SPLINE
SPL {X  -162.820, Y  +621.304, Z    +0.000, E1   +22.259, E3 +517644.135}
SPL {X  -162.820, Y  +618.758, Z    +0.000, E1   +22.239, E3 +517657.285}
SPL {X  -162.820, Y  +616.062, Z    +0.000, E1   +22.275, E3 +517670.706}
SPL {X  -162.820, Y  +613.536, Z    +0.000, E1   +22.242, E3 +517683.827}
SPL {X  -162.820, Y  +611.128, Z    +0.000, E1   +22.252, E3 +517695.998}
SPL {X  -162.820, Y  +608.428, Z    +0.000, E1   +22.255, E3 +517709.782}
SPL {X  -162.820, Y  +605.178, Z    +0.000, E1   +22.267, E3 +517726.314}
SPL {X  -162.820, Y  +602.350, Z    +0.000, E1   +22.224, E3 +517740.931}
SPL {X  -162.820, Y  +599.168, Z    +0.000, E1   +22.310, E3 +517756.585}
SPL {X  -162.820, Y  +595.597, Z    +0.000, E1   +22.284, E3 +517774.921}
SPL {X  -162.820, Y  +593.320, Z    +0.000, E1   +22.199, E3 +517787.011}
SPL {X  -162.820, Y  +591.031, Z    +0.000, E1   +22.283, E3 +517798.102}
SPL {X  -162.820, Y  +588.026, Z    +0.000, E1   +22.301, E3 +517813.229}
SPL {X  -162.820, Y  +585.899, Z    +0.000, E1   +22.286, E3 +517824.031}
SPL {X  -162.820, Y  +583.204, Z    +0.000, E1   +22.278, E3 +517838.054}
SPL {X  -162.820, Y  +580.317, Z    +0.000, E1   +22.300, E3 +517852.325}
SPL {X  -162.820, Y  +578.061, Z    +0.000, E1   +22.264, E3 +517864.210}
SPL {X  -162.820, Y  +575.394, Z    +0.000, E1   +22.240, E3 +517877.954}
SPL {X  -162.820, Y  +573.156, Z    +0.000, E1   +22.254, E3 +517889.164}
SPL {X  -162.820, Y  +570.852, Z    +0.000, E1   +22.234, E3 +517901.188}
SPL {X  -162.820, Y  +568.608, Z    +0.000, E1   +22.253, E3 +517912.321}
SPL {X  -162.820, Y  +565.838, Z    +0.000, E1   +22.271, E3 +517926.553}
SPL {X  -162.820, Y  +562.162, Z    +0.000, E1   +22.252, E3 +517945.370}
SPL {X  -162.820, Y  +559.515, Z    +0.000, E1   +22.273, E3 +517958.488}
SPL {X  -162.820, Y  +556.723, Z    +0.000, E1   +22.309, E3 +517972.572}
SPL {X  -162.820, Y  +553.294, Z    +0.000, E1   +22.266, E3 +517990.360}
SPL {X  -162.820, Y  +550.136, Z    +0.000, E1   +22.258, E3 +518006.473}
SPL {X  -162.820, Y  +546.694, Z    +0.000, E1   +22.290, E3 +518023.795}
SPL {X  -162.820, Y  +543.558, Z    +0.000, E1   +22.285, E3 +518039.658}
SPL {X  -162.820, Y  +541.633, Z    +0.000, E1   +22.257, E3 +518049.586}
SPL {X  -162.820, Y  +539.116, Z    +0.000, E1   +22.302, E3 +518062.197}
SPL {X  -162.820, Y  +536.913, Z    +0.000, E1   +22.192, E3 +518074.121}
SPL {X  -162.820, Y  +534.880, Z    +0.000, E1   +22.252, E3 +518084.075}
SPL {X  -162.820, Y  +532.896, Z    +0.000, E1   +22.234, E3 +518094.235}
SPL {X  -162.820, Y  +531.056, Z    +0.000, E1   +22.251, E3 +518103.517}
SPL {X  -162.820, Y  +528.708, Z    +0.000, E1   +22.319, E3 +518114.899}
SPL {X  -162.820, Y  +525.932, Z    +0.000, E1   +22.258, E3 +518129.655}
SPL {X  -162.820, Y  +522.524, Z    +0.000, E1   +22.326, E3 +518146.379}
SPL {X  -162.820, Y  +519.457, Z    +0.000, E1   +22.481, E3 +518160.508}
SPL {X  -162.820, Y  +505.859, Z    +0.000, E1   +28.367, E3 +518174.991}
SPL {X  -162.820, Y  +504.131, Z    +0.000, E1   +27.325, E3 +518189.129}
SPL {X  -162.820, Y  +503.215, Z    +0.000, E1   +26.369, E3 +518199.815}
SPL {X  -162.820, Y  +502.502, Z    +0.000, E1   +25.597, E3 +518208.662}
SPL {X  -162.820, Y  +501.672, Z    +0.000, E1   +24.583, E3 +518220.277}
SPL {X  -162.820, Y  +500.515, Z    +0.000, E1   +23.444, E3 +518234.807}
SPL {X  -162.820, Y  +499.633, Z    +0.000, E1   +22.486, E3 +518246.853}
SPL {X  -162.820, Y  +498.303, Z    +0.000, E1   +21.749, E3 +518260.163}
SPL {X  -162.820, Y  +495.897, Z    +0.000, E1   +21.662, E3 +518273.316}
SPL {X  -162.820, Y  +493.717, Z    +0.000, E1   +21.704, E3 +518284.422}
SPL {X  -162.820, Y  +491.396, Z    +0.000, E1   +21.707, E3 +518296.546}
SPL {X  -162.820, Y  +489.485, Z    +0.000, E1   +21.661, E3 +518306.894}
SPL {X  -162.820, Y  +487.723, Z    +0.000, E1   +21.665, E3 +518316.098}
SPL {X  -162.820, Y  +485.661, Z    +0.000, E1   +21.712, E3 +518326.541}
SPL {X  -162.820, Y  +482.775, Z    +0.000, E1   +21.716, E3 +518341.794}
SPL {X  -162.820, Y  +479.894, Z    +0.000, E1   +21.695, E3 +518356.870}
SPL {X  -162.820, Y  +477.685, Z    +0.000, E1   +21.656, E3 +518368.807}
SPL {X  -162.820, Y  +475.419, Z    +0.000, E1   +21.711, E3 +518380.160}
SPL {X  -162.820, Y  +473.301, Z    +0.000, E1   +21.712, E3 +518391.257}
SPL {X  -162.820, Y  +470.965, Z    +0.000, E1   +21.700, E3 +518403.602}
SPL {X  -162.820, Y  +469.036, Z    +0.000, E1   +21.695, E3 +518413.646}
SPL {X  -162.820, Y  +467.138, Z    +0.000, E1   +21.678, E3 +518423.817}
SPL {X  -162.820, Y  +465.011, Z    +0.000, E1   +21.692, E3 +518434.800}
SPL {X  -162.820, Y  +462.669, Z    +0.000, E1   +21.752, E3 +518446.580}
SPL {X  -162.820, Y  +460.725, Z    +0.000, E1   +21.689, E3 +518457.193}
SPL {X  -162.820, Y  +458.666, Z    +0.000, E1   +21.695, E3 +518468.005}
SPL {X  -162.820, Y  +456.431, Z    +0.000, E1   +21.708, E3 +518479.534}
SPL {X  -162.820, Y  +454.628, Z    +0.000, E1   +21.674, E3 +518489.252}
SPL {X  -162.820, Y  +452.690, Z    +0.000, E1   +21.773, E3 +518498.526}
SPL {X  -162.820, Y  +450.610, Z    +0.000, E1   +21.698, E3 +518510.125}
SPL {X  -162.820, Y  +448.170, Z    +0.000, E1   +21.667, E3 +518523.146}
SPL {X  -162.820, Y  +446.246, Z    +0.000, E1   +21.696, E3 +518532.964}
SPL {X  -162.820, Y  +443.784, Z    +0.000, E1   +21.713, E3 +518545.750}
SPL {X  -162.820, Y  +441.754, Z    +0.000, E1   +21.708, E3 +518556.302}
SPL {X  -162.820, Y  +439.933, Z    +0.000, E1   +21.690, E3 +518566.066}
SPL {X  -162.820, Y  +437.628, Z    +0.000, E1   +21.678, E3 +518578.254}
SPL {X  -162.820, Y  +434.473, Z    +0.000, E1   +21.747, E3 +518594.350}
SPL {X  -162.820, Y  +431.492, Z    +0.000, E1   +21.686, E3 +518610.299}
SPL {X  -162.820, Y  +429.074, Z    +0.000, E1   +21.710, E3 +518622.751}
SPL {X  -162.820, Y  +426.023, Z    +0.000, E1   +21.718, E3 +518638.819}
SPL {X  -162.820, Y  +422.986, Z    +0.000, E1   +21.685, E3 +518654.866}
SPL {X  -162.820, Y  +420.528, Z    +0.000, E1   +21.706, E3 +518667.516}
SPL {X  -162.820, Y  +418.116, Z    +0.000, E1   +21.761, E3 +518679.663}
SPL {X  -162.820, Y  +416.127, Z    +0.000, E1   +21.715, E3 +518690.368}
SPL {X  -162.820, Y  +414.361, Z    +0.000, E1   +21.613, E3 +518700.556}
SPL {X  -162.820, Y  +411.450, Z    +0.000, E1   +21.710, E3 +518715.129}
SPL {X  -162.820, Y  +408.590, Z    +0.000, E1   +21.735, E3 +518729.755}
SPL {X  -162.820, Y  +406.238, Z    +0.000, E1   +21.697, E3 +518742.404}
SPL {X  -162.820, Y  +403.166, Z    +0.000, E1   +21.746, E3 +518758.209}
SPL {X  -162.820, Y  +400.348, Z    +0.000, E1   +21.713, E3 +518773.044}
SPL {X  -162.820, Y  +398.298, Z    +0.000, E1   +21.721, E3 +518783.660}
SPL {X  -162.820, Y  +396.371, Z    +0.000, E1   +21.713, E3 +518793.842}
SPL {X  -162.820, Y  +394.508, Z    +0.000, E1   +21.616, E3 +518804.397}
SPL {X  -162.820, Y  +391.777, Z    +0.000, E1   +21.714, E3 +518818.057}
SPL {X  -162.820, Y  +388.822, Z    +0.000, E1   +21.717, E3 +518833.376}
SPL {X  -162.820, Y  +386.818, Z    +0.000, E1   +21.679, E3 +518844.116}
SPL {X  -162.820, Y  +384.697, Z    +0.000, E1   +21.693, E3 +518855.186}
SPL {X  -162.820, Y  +382.288, Z    +0.000, E1   +21.742, E3 +518867.310}
SPL {X  -162.817, Y  +379.520, Z    +0.000, E1   +21.723, E3 +518882.147}
SPL {X  -162.776, Y  +376.710, Z    +0.000, E1   +21.698, E3 +518896.887}
SPL {X  -162.707, Y  +374.438, Z    +0.000, E1   +21.688, E3 +518908.890}
SPL {X  -162.607, Y  +372.171, Z    +0.000, E1   +21.692, E3 +518920.690}
SPL {X  -162.494, Y  +370.197, Z    +0.000, E1   +21.655, E3 +518931.316}
SPL {X  -162.349, Y  +368.131, Z    +0.000, E1   +21.624, E3 +518942.434}
SPL {X  -162.161, Y  +365.866, Z    +0.000, E1   +21.642, E3 +518954.120}
SPL {X  -161.927, Y  +363.466, Z    +0.000, E1   +21.730, E3 +518965.891}
SPL {X  -160.290, Y  +351.907, Z    +0.000, E1   +27.562, E3 +518973.469}
SPL {X  -159.725, Y  +348.905, Z    +0.000, E1   +26.136, E3 +518998.704}
ENDSPLINE

SPLINE
SPL {X  -160.871, Y  +355.385, Z    +0.000, E1   +21.841, E3 +519007.547}
SPL {X  -161.833, Y  +362.603, Z    +0.000, E1   +17.021, E3 +519017.578}
ENDSPLINE

SPLINE
SPL {X  -160.786, Y  +354.842, Z    +0.000, E1   +19.274, E3 +519049.733}
ENDSPLINE

SPLINE
SPL {X  -162.485, Y  +370.062, Z    +0.000, E1   +10.606, E3 +519056.111}
SPL {X  -162.818, Y  +379.636, Z    +0.000, E1    +5.115, E3 +519045.460}
SPL {X  -162.820, Y  +386.976, Z    +0.000, E1    +0.144, E3 +519044.559}
SPL {X  -162.820, Y  +391.982, Z    +0.000, E1    -3.443, E3 +519051.324}
SPL {X  -162.820, Y  +399.630, Z    +0.000, E1    -9.426, E3 +519053.832}
SPL {X  -162.820, Y  +408.127, Z    +0.000, E1   -18.417, E3 +519040.120}
SPL {X  -162.820, Y  +420.083, Z    +0.000, E1   -24.325, E3 +519060.596}
SPL {X  -162.820, Y  +428.527, Z    +0.000, E1   -26.988, E3 +519077.888}
SPL {X  -162.820, Y  +431.191, Z    +0.000, E1   -23.548, E3 +519112.741}
SPL {X  -162.820, Y  +432.946, Z    +0.000, E1   -22.795, E3 +519127.144}
SPL {X  -162.820, Y  +434.888, Z    +0.000, E1   -22.823, E3 +519136.551}
SPL {X  -162.820, Y  +436.834, Z    +0.000, E1   -22.779, E3 +519146.511}
SPL {X  -162.820, Y  +438.868, Z    +0.000, E1   -22.837, E3 +519156.165}
SPL {X  -162.820, Y  +441.351, Z    +0.000, E1   -22.805, E3 +519168.740}
SPL {X  -162.820, Y  +443.809, Z    +0.000, E1   -22.804, E3 +519180.906}
SPL {X  -162.820, Y  +446.105, Z    +0.000, E1   -22.815, E3 +519192.148}
SPL {X  -162.820, Y  +447.974, Z    +0.000, E1   -22.856, E3 +519201.051}
SPL {X  -162.820, Y  +449.911, Z    +0.000, E1   -22.774, E3 +519211.326}
SPL {X  -162.820, Y  +451.861, Z    +0.000, E1   -22.750, E3 +519221.173}
SPL {X  -162.820, Y  +454.167, Z    +0.000, E1   -22.842, E3 +519231.903}
SPL {X  -162.820, Y  +456.529, Z    +0.000, E1   -22.855, E3 +519243.431}
SPL {X  -162.820, Y  +458.725, Z    +0.000, E1   -22.793, E3 +519254.836}
SPL {X  -162.820, Y  +460.754, Z    +0.000, E1   -22.806, E3 +519264.709}
SPL {X  -162.820, Y  +462.409, Z    +0.000, E1   -22.783, E3 +519273.126}
SPL {X  -162.820, Y  +464.633, Z    +0.000, E1   -22.813, E3 +519283.955}
SPL {X  -162.820, Y  +467.913, Z    +0.000, E1   -22.879, E3 +519299.794}
SPL {X  -162.820, Y  +470.892, Z    +0.000, E1   -22.837, E3 +519314.684}
SPL {X  -162.820, Y  +472.726, Z    +0.000, E1   -22.777, E3 +519324.222}
SPL {X  -162.820, Y  +475.118, Z    +0.000, E1   -22.777, E3 +519336.194}
SPL {X  -162.820, Y  +477.389, Z    +0.000, E1   -22.803, E3 +519347.110}
SPL {X  -162.820, Y  +478.914, Z    +0.000, E1   -22.821, E3 +519354.502}
SPL {X  -162.820, Y  +481.034, Z    +0.000, E1   -22.831, E3 +519365.024}
SPL {X  -162.820, Y  +484.256, Z    +0.000, E1   -22.840, E3 +519381.043}
SPL {X  -162.820, Y  +487.952, Z    +0.000, E1   -22.824, E3 +519399.473}
SPL {X  -162.820, Y  +491.768, Z    +0.000, E1   -22.852, E3 +519418.154}
SPL {X  -162.820, Y  +495.526, Z    +0.000, E1   -22.833, E3 +519436.925}
SPL {X  -162.820, Y  +499.330, Z    +0.000, E1   -22.841, E3 +519455.706}
SPL {X  -162.820, Y  +503.049, Z    +0.000, E1   -22.823, E3 +519474.255}
SPL {X  -162.820, Y  +506.908, Z    +0.000, E1   -22.877, E3 +519492.925}
SPL {X  -162.820, Y  +510.068, Z    +0.000, E1   -22.761, E3 +519509.397}
SPL {X  -162.820, Y  +512.359, Z    +0.000, E1   -22.823, E3 +519520.129}
SPL {X  -162.820, Y  +513.873, Z    +0.000, E1   -22.800, E3 +519527.815}
SPL {X  -162.820, Y  +516.100, Z    +0.000, E1   -22.809, E3 +519538.892}
SPL {X  -162.820, Y  +518.662, Z    +0.000, E1   -22.847, E3 +519551.190}
SPL {X  -162.820, Y  +520.641, Z    +0.000, E1   -22.790, E3 +519561.431}
SPL {X  -162.820, Y  +523.535, Z    +0.000, E1   -22.857, E3 +519575.400}
SPL {X  -162.820, Y  +526.661, Z    +0.000, E1   -22.801, E3 +519591.224}
SPL {X  -162.820, Y  +528.725, Z    +0.000, E1   -22.770, E3 +519601.594}
SPL {X  -162.820, Y  +530.303, Z    +0.000, E1   -22.798, E3 +519609.213}
SPL {X  -162.820, Y  +532.614, Z    +0.000, E1   -22.828, E3 +519620.481}
SPL {X  -162.820, Y  +534.838, Z    +0.000, E1   -22.864, E3 +519631.110}
SPL {X  -162.820, Y  +536.882, Z    +0.000, E1   -22.782, E3 +519641.965}
SPL {X  -162.820, Y  +539.194, Z    +0.000, E1   -22.826, E3 +519653.013}
SPL {X  -162.820, Y  +541.555, Z    +0.000, E1   -22.817, E3 +519664.828}
SPL {X  -162.820, Y  +543.728, Z    +0.000, E1   -22.799, E3 +519675.685}
SPL {X  -162.820, Y  +545.925, Z    +0.000, E1   -22.803, E3 +519686.555}
SPL {X  -162.820, Y  +549.071, Z    +0.000, E1   -22.836, E3 +519702.083}
SPL {X  -162.820, Y  +553.089, Z    +0.000, E1   -22.838, E3 +519721.983}
SPL {X  -162.820, Y  +556.430, Z    +0.000, E1   -22.821, E3 +519738.484}
SPL {X  -162.820, Y  +558.974, Z    +0.000, E1   -22.806, E3 +519751.184}
SPL {X  -162.820, Y  +562.171, Z    +0.000, E1   -22.845, E3 +519766.882}
SPL {X  -162.820, Y  +565.170, Z    +0.000, E1   -22.801, E3 +519781.895}
SPL {X  -162.820, Y  +567.308, Z    +0.000, E1   -22.750, E3 +519792.911}
SPL {X  -162.820, Y  +570.378, Z    +0.000, E1   -22.843, E3 +519807.535}
SPL {X  -162.820, Y  +573.634, Z    +0.000, E1   -22.827, E3 +519823.679}
SPL {X  -162.820, Y  +576.228, Z    +0.000, E1   -22.814, E3 +519836.575}
SPL {X  -162.820, Y  +578.553, Z    +0.000, E1   -22.801, E3 +519848.191}
SPL {X  -162.820, Y  +581.064, Z    +0.000, E1   -22.823, E3 +519860.476}
SPL {X  -162.820, Y  +583.435, Z    +0.000, E1   -22.808, E3 +519872.297}
SPL {X  -162.820, Y  +585.410, Z    +0.000, E1   -22.764, E3 +519882.433}
SPL {X  -162.820, Y  +587.676, Z    +0.000, E1   -22.853, E3 +519892.948}
SPL {X  -162.820, Y  +589.682, Z    +0.000, E1   -22.776, E3 +519903.477}
SPL {X  -162.820, Y  +591.720, Z    +0.000, E1   -22.868, E3 +519912.788}
SPL {X  -162.820, Y  +593.650, Z    +0.000, E1   -22.810, E3 +519922.858}
SPL {X  -162.820, Y  +595.830, Z    +0.000, E1   -22.828, E3 +519933.474}
SPL {X  -162.820, Y  +598.094, Z    +0.000, E1   -22.843, E3 +519944.587}
SPL {X  -162.820, Y  +600.420, Z    +0.000, E1   -22.826, E3 +519956.218}
SPL {X  -162.820, Y  +602.573, Z    +0.000, E1   -22.830, E3 +519966.803}
SPL {X  -162.820, Y  +604.828, Z    +0.000, E1   -22.784, E3 +519978.442}
SPL {X  -162.820, Y  +607.142, Z    +0.000, E1   -22.808, E3 +519989.623}
SPL {X  -162.820, Y  +608.890, Z    +0.000, E1   -22.790, E3 +519998.447}
SPL {X  -162.820, Y  +611.103, Z    +0.000, E1   -22.785, E3 +520009.485}
SPL {X  -162.820, Y  +613.294, Z    +0.000, E1   -22.780, E3 +520020.358}
SPL {X  -162.820, Y  +615.356, Z    +0.000, E1   -22.799, E3 +520030.416}
SPL {X  -162.820, Y  +617.439, Z    +0.000, E1   -22.808, E3 +520040.674}
SPL {X  -162.820, Y  +619.665, Z    +0.000, E1   -22.817, E3 +520051.642}
SPL {X  -162.820, Y  +621.733, Z    +0.000, E1   -22.759, E3 +520062.366}
SPL {X  -162.820, Y  +624.076, Z    +0.000, E1   -22.774, E3 +520073.871}
SPL {X  -162.820, Y  +627.244, Z    +0.000, E1   -22.803, E3 +520089.553}
SPL {X  -162.820, Y  +630.349, Z    +0.000, E1   -22.766, E3 +520105.085}
SPL {X  -162.820, Y  +632.572, Z    +0.000, E1   -22.785, E3 +520115.892}
SPL {X  -162.820, Y  +634.507, Z    +0.000, E1   -22.784, E3 +520125.531}
SPL {X  -162.820, Y  +636.863, Z    +0.000, E1   -22.760, E3 +520137.453}
SPL {X  -162.820, Y  +640.111, Z    +0.000, E1   -22.809, E3 +520153.336}
SPL {X  -162.820, Y  +643.449, Z    +0.000, E1   -22.796, E3 +520169.853}
SPL {X  -162.820, Y  +645.630, Z    +0.000, E1   -22.795, E3 +520180.549}
SPL {X  -162.820, Y  +647.561, Z    +0.000, E1   -22.705, E3 +520191.000}
SPL {X  -162.820, Y  +649.758, Z    +0.000, E1   -22.780, E3 +520201.190}
SPL {X  -162.820, Y  +651.708, Z    +0.000, E1   -22.810, E3 +520210.685}
SPL {X  -162.820, Y  +653.898, Z    +0.000, E1   -22.796, E3 +520221.605}
SPL {X  -162.820, Y  +656.161, Z    +0.000, E1   -22.812, E3 +520232.727}
SPL {X  -162.820, Y  +658.384, Z    +0.000, E1   -22.822, E3 +520243.593}
SPL {X  -162.820, Y  +660.215, Z    +0.000, E1   -22.649, E3 +520254.184}
SPL {X  -162.820, Y  +662.823, Z    +0.000, E1   -22.799, E3 +520265.892}
SPL {X  -162.820, Y  +665.862, Z    +0.000, E1   -22.864, E3 +520280.591}
SPL {X  -162.820, Y  +668.960, Z    +0.000, E1   -22.773, E3 +520296.542}
SPL {X  -162.820, Y  +671.605, Z    +0.000, E1   -22.777, E3 +520309.616}
SPL {X  -162.817, Y  +674.515, Z    +0.000, E1   -22.816, E3 +520323.813}
SPL {X  -162.773, Y  +677.428, Z    +0.000, E1   -22.762, E3 +520338.621}
SPL {X  -162.691, Y  +679.987, Z    +0.000, E1   -22.794, E3 +520351.034}
SPL {X  -162.604, Y  +681.880, Z    +0.000, E1   -22.691, E3 +520361.195}
SPL {X  -162.458, Y  +684.346, Z    +0.000, E1   -22.764, E3 +520372.988}
SPL {X  -162.229, Y  +687.364, Z    +0.000, E1   -22.685, E3 +520388.608}
SPL {X  -161.938, Y  +690.422, Z    +0.000, E1   -22.769, E3 +520403.014}
SPL {X  -161.065, Y  +697.344, Z    +0.000, E1   -25.698, E3 +520412.134}
SPL {X  -158.553, Y  +710.529, Z    +0.000, E1   -30.890, E3 +520426.030}
ENDSPLINE

SPLINE
SPL {X  -161.215, Y  +696.305, Z    +0.000, E1   -20.575, E3 +520452.611}
SPL {X  -161.691, Y  +692.643, Z    +0.000, E1   -17.369, E3 +520468.799}
SPL {X  -162.534, Y  +683.153, Z    +0.000, E1   -10.475, E3 +520494.266}
SPL {X  -162.820, Y  +667.630, Z    +0.000, E1    -0.882, E3 +520488.243}
SPL {X  -162.820, Y  +661.883, Z    +0.000, E1    +3.373, E3 +520493.686}
SPL {X  -162.820, Y  +655.163, Z    +0.000, E1    +8.702, E3 +520493.285}
SPL {X  -162.820, Y  +634.515, Z    +0.000, E1   +26.439, E3 +520485.698}
ENDSPLINE

SPLINE
SPL {X  -162.820, Y  +638.080, Z    +0.000, E1   +18.858, E3 +520515.662}
ENDSPLINE

SPLINE
SPL {X  -162.820, Y  +623.278, Z    +0.000, E1   +28.723, E3 +520517.233}
SPL {X  -162.820, Y  +611.829, Z    +0.000, E1   +31.229, E3 +520540.885}
ENDSPLINE

SPLINE
SPL {X  -162.820, Y  +623.595, Z    +0.000, E1   +22.712, E3 +520555.806}
ENDSPLINE

SPLINE
SPL {X  -162.820, Y  +621.304, Z    +0.000, E1   +22.259, E3 +520570.964}
SPL {X  -162.820, Y  +618.758, Z    +0.000, E1   +22.239, E3 +520584.115}
SPL {X  -162.820, Y  +616.062, Z    +0.000, E1   +22.275, E3 +520597.535}
SPL {X  -162.820, Y  +613.536, Z    +0.000, E1   +22.242, E3 +520610.657}
SPL {X  -162.820, Y  +610.461, Z    +0.000, E1   +22.264, E3 +520626.288}
SPL {X  -162.820, Y  +606.755, Z    +0.000, E1   +22.275, E3 +520645.086}
SPL {X  -162.820, Y  +603.020, Z    +0.000, E1   +22.272, E3 +520664.146}
SPL {X  -162.820, Y  +599.842, Z    +0.000, E1   +22.298, E3 +520679.912}
SPL {X  -162.820, Y  +597.194, Z    +0.000, E1   +22.253, E3 +520693.833}
SPL {X  -162.820, Y  +594.779, Z    +0.000, E1   +22.284, E3 +520705.737}
SPL {X  -162.820, Y  +592.389, Z    +0.000, E1   +22.245, E3 +520718.353}
SPL {X  -162.820, Y  +589.492, Z    +0.000, E1   +22.304, E3 +520732.537}
SPL {X  -162.820, Y  +587.447, Z    +0.000, E1   +22.279, E3 +520743.066}
SPL {X  -162.820, Y  +585.192, Z    +0.000, E1   +22.298, E3 +520754.477}
SPL {X  -162.820, Y  +582.610, Z    +0.000, E1   +22.234, E3 +520768.100}
SPL {X  -162.820, Y  +579.691, Z    +0.000, E1   +22.312, E3 +520782.371}
SPL {X  -162.820, Y  +577.460, Z    +0.000, E1   +22.218, E3 +520794.358}
SPL {X  -162.820, Y  +575.394, Z    +0.000, E1   +22.240, E3 +520804.783}
SPL {X  -162.820, Y  +572.645, Z    +0.000, E1   +22.246, E3 +520818.781}
SPL {X  -162.820, Y  +570.282, Z    +0.000, E1   +22.231, E3 +520830.831}
SPL {X  -162.820, Y  +567.961, Z    +0.000, E1   +22.247, E3 +520842.621}
SPL {X  -162.820, Y  +565.204, Z    +0.000, E1   +22.256, E3 +520856.564}
SPL {X  -162.820, Y  +562.162, Z    +0.000, E1   +22.252, E3 +520872.199}
SPL {X  -162.820, Y  +558.919, Z    +0.000, E1   +22.286, E3 +520888.362}
SPL {X  -162.820, Y  +556.169, Z    +0.000, E1   +22.295, E3 +520902.192}
SPL {X  -162.820, Y  +553.294, Z    +0.000, E1   +22.266, E3 +520917.189}
SPL {X  -162.820, Y  +550.136, Z    +0.000, E1   +22.258, E3 +520933.302}
SPL {X  -162.820, Y  +547.491, Z    +0.000, E1   +22.292, E3 +520946.345}
SPL {X  -162.820, Y  +545.860, Z    +0.000, E1   +22.216, E3 +520955.257}
SPL {X  -162.820, Y  +543.558, Z    +0.000, E1   +22.285, E3 +520966.487}
SPL {X  -162.820, Y  +540.968, Z    +0.000, E1   +22.274, E3 +520979.760}
SPL {X  -162.820, Y  +538.512, Z    +0.000, E1   +22.287, E3 +520992.072}
SPL {X  -162.820, Y  +535.523, Z    +0.000, E1   +22.266, E3 +521007.688}
SPL {X  -162.820, Y  +531.757, Z    +0.000, E1   +22.276, E3 +521026.742}
SPL {X  -162.820, Y  +527.980, Z    +0.000, E1   +22.326, E3 +521045.573}
SPL {X  -162.820, Y  +524.599, Z    +0.000, E1   +22.287, E3 +521062.971}
SPL {X  -162.820, Y  +522.011, Z    +0.000, E1   +22.282, E3 +521076.048}
SPL {X  -162.820, Y  +519.457, Z    +0.000, E1   +22.481, E3 +521087.337}
SPL {X  -162.820, Y  +505.859, Z    +0.000, E1   +28.367, E3 +521101.820}
SPL {X  -162.820, Y  +504.131, Z    +0.000, E1   +27.325, E3 +521115.958}
SPL {X  -162.820, Y  +502.813, Z    +0.000, E1   +26.013, E3 +521131.335}
SPL {X  -162.820, Y  +502.016, Z    +0.000, E1   +24.802, E3 +521143.677}
SPL {X  -162.820, Y  +501.060, Z    +0.000, E1   +24.081, E3 +521153.867}
SPL {X  -162.820, Y  +500.336, Z    +0.000, E1   +23.110, E3 +521165.007}
SPL {X  -162.820, Y  +499.240, Z    +0.000, E1   +22.316, E3 +521177.318}
SPL {X  -162.820, Y  +498.027, Z    +0.000, E1   +21.516, E3 +521190.225}
SPL {X  -162.820, Y  +495.897, Z    +0.000, E1   +21.662, E3 +521200.145}
SPL {X  -162.820, Y  +493.717, Z    +0.000, E1   +21.704, E3 +521211.252}
SPL {X  -162.820, Y  +491.396, Z    +0.000, E1   +21.707, E3 +521223.376}
SPL {X  -162.820, Y  +488.560, Z    +0.000, E1   +21.695, E3 +521238.485}
SPL {X  -162.820, Y  +485.661, Z    +0.000, E1   +21.712, E3 +521253.370}
SPL {X  -162.820, Y  +482.775, Z    +0.000, E1   +21.716, E3 +521268.623}
SPL {X  -162.820, Y  +479.894, Z    +0.000, E1   +21.695, E3 +521283.699}
SPL {X  -162.820, Y  +477.685, Z    +0.000, E1   +21.656, E3 +521295.637}
SPL {X  -162.820, Y  +475.419, Z    +0.000, E1   +21.711, E3 +521306.989}
SPL {X  -162.820, Y  +473.301, Z    +0.000, E1   +21.712, E3 +521318.086}
SPL {X  -162.820, Y  +470.965, Z    +0.000, E1   +21.700, E3 +521330.431}
SPL {X  -162.820, Y  +469.036, Z    +0.000, E1   +21.695, E3 +521340.475}
SPL {X  -162.820, Y  +467.138, Z    +0.000, E1   +21.678, E3 +521350.647}
SPL {X  -162.820, Y  +465.011, Z    +0.000, E1   +21.692, E3 +521361.629}
SPL {X  -162.820, Y  +462.669, Z    +0.000, E1   +21.752, E3 +521373.410}
SPL {X  -162.820, Y  +460.725, Z    +0.000, E1   +21.689, E3 +521384.023}
SPL {X  -162.820, Y  +458.666, Z    +0.000, E1   +21.695, E3 +521394.835}
SPL {X  -162.820, Y  +456.431, Z    +0.000, E1   +21.708, E3 +521406.363}
SPL {X  -162.820, Y  +453.609, Z    +0.000, E1   +21.757, E3 +521420.897}
SPL {X  -162.820, Y  +450.610, Z    +0.000, E1   +21.698, E3 +521436.954}
SPL {X  -162.820, Y  +448.170, Z    +0.000, E1   +21.667, E3 +521449.975}
SPL {X  -162.820, Y  +446.246, Z    +0.000, E1   +21.696, E3 +521459.793}
SPL {X  -162.820, Y  +443.784, Z    +0.000, E1   +21.713, E3 +521472.579}
SPL {X  -162.820, Y  +440.567, Z    +0.000, E1   +21.731, E3 +521489.419}
SPL {X  -162.820, Y  +437.628, Z    +0.000, E1   +21.678, E3 +521505.083}
SPL {X  -162.820, Y  +434.473, Z    +0.000, E1   +21.747, E3 +521521.179}
SPL {X  -162.820, Y  +431.492, Z    +0.000, E1   +21.686, E3 +521537.128}
SPL {X  -162.820, Y  +429.074, Z    +0.000, E1   +21.710, E3 +521549.580}
SPL {X  -162.820, Y  +426.023, Z    +0.000, E1   +21.718, E3 +521565.648}
SPL {X  -162.820, Y  +422.986, Z    +0.000, E1   +21.685, E3 +521581.695}
SPL {X  -162.820, Y  +420.528, Z    +0.000, E1   +21.706, E3 +521594.345}
SPL {X  -162.820, Y  +418.116, Z    +0.000, E1   +21.761, E3 +521606.492}
SPL {X  -162.820, Y  +416.127, Z    +0.000, E1   +21.715, E3 +521617.198}
SPL {X  -162.820, Y  +414.361, Z    +0.000, E1   +21.613, E3 +521627.385}
SPL {X  -162.820, Y  +411.450, Z    +0.000, E1   +21.710, E3 +521641.958}
SPL {X  -162.820, Y  +408.590, Z    +0.000, E1   +21.735, E3 +521656.584}
SPL {X  -162.820, Y  +406.238, Z    +0.000, E1   +21.697, E3 +521669.233}
SPL {X  -162.820, Y  +403.166, Z    +0.000, E1   +21.746, E3 +521685.039}
SPL {X  -162.820, Y  +400.348, Z    +0.000, E1   +21.713, E3 +521699.874}
SPL {X  -162.820, Y  +398.298, Z    +0.000, E1   +21.721, E3 +521710.489}
SPL {X  -162.820, Y  +396.371, Z    +0.000, E1   +21.713, E3 +521720.671}
SPL {X  -162.820, Y  +394.508, Z    +0.000, E1   +21.616, E3 +521731.226}
SPL {X  -162.820, Y  +391.777, Z    +0.000, E1   +21.714, E3 +521744.886}
SPL {X  -162.820, Y  +388.822, Z    +0.000, E1   +21.717, E3 +521760.205}
SPL {X  -162.820, Y  +386.818, Z    +0.000, E1   +21.679, E3 +521770.945}
SPL {X  -162.820, Y  +384.697, Z    +0.000, E1   +21.693, E3 +521782.016}
SPL {X  -162.820, Y  +382.288, Z    +0.000, E1   +21.742, E3 +521794.139}
SPL {X  -162.817, Y  +379.520, Z    +0.000, E1   +21.723, E3 +521808.977}
SPL {X  -162.776, Y  +376.710, Z    +0.000, E1   +21.698, E3 +521823.716}
SPL {X  -162.707, Y  +374.438, Z    +0.000, E1   +21.688, E3 +521835.720}
SPL {X  -162.607, Y  +372.171, Z    +0.000, E1   +21.692, E3 +521847.519}
SPL {X  -162.494, Y  +370.197, Z    +0.000, E1   +21.655, E3 +521858.146}
SPL {X  -162.349, Y  +368.131, Z    +0.000, E1   +21.624, E3 +521869.264}
SPL {X  -162.161, Y  +365.866, Z    +0.000, E1   +21.642, E3 +521880.949}
SPL {X  -161.651, Y  +361.024, Z    +0.000, E1   +22.970, E3 +521894.372}
SPL {X  -160.281, Y  +351.857, Z    +0.000, E1   +24.243, E3 +521929.711}
ENDSPLINE

SPLINE
SPL {X  -161.833, Y  +362.603, Z    +0.000, E1   +17.021, E3 +521944.407}
ENDSPLINE

SPLINE
SPL {X  -160.786, Y  +354.842, Z    +0.000, E1   +19.274, E3 +521976.563}
ENDSPLINE

SPLINE
SPL {X  -162.485, Y  +370.062, Z    +0.000, E1   +10.606, E3 +521982.941}
SPL {X  -162.820, Y  +381.311, Z    +0.000, E1    +4.054, E3 +521973.296}
SPL {X  -162.820, Y  +389.994, Z    +0.000, E1    -2.149, E3 +521967.708}
SPL {X  -162.820, Y  +391.982, Z    +0.000, E1    -3.443, E3 +521978.154}
SPL {X  -162.820, Y  +399.630, Z    +0.000, E1    -9.426, E3 +521980.661}
SPL {X  -162.820, Y  +408.127, Z    +0.000, E1   -18.417, E3 +521966.949}
SPL {X  -162.820, Y  +420.083, Z    +0.000, E1   -24.325, E3 +521987.425}
SPL {X  -162.820, Y  +428.527, Z    +0.000, E1   -26.988, E3 +522004.717}
SPL {X  -162.820, Y  +431.336, Z    +0.000, E1   -24.162, E3 +522034.927}
SPL {X  -162.820, Y  +432.048, Z    +0.000, E1   -22.832, E3 +522049.431}
SPL {X  -162.820, Y  +434.888, Z    +0.000, E1   -22.823, E3 +522063.380}
SPL {X  -162.820, Y  +436.834, Z    +0.000, E1   -22.779, E3 +522073.340}
SPL {X  -162.820, Y  +438.868, Z    +0.000, E1   -22.837, E3 +522082.994}
SPL {X  -162.820, Y  +441.351, Z    +0.000, E1   -22.805, E3 +522095.569}
SPL {X  -162.820, Y  +443.809, Z    +0.000, E1   -22.804, E3 +522107.735}
SPL {X  -162.820, Y  +446.105, Z    +0.000, E1   -22.815, E3 +522118.978}
SPL {X  -162.820, Y  +447.974, Z    +0.000, E1   -22.856, E3 +522127.880}
SPL {X  -162.820, Y  +449.911, Z    +0.000, E1   -22.774, E3 +522138.155}
SPL {X  -162.820, Y  +451.861, Z    +0.000, E1   -22.750, E3 +522148.003}
SPL {X  -162.820, Y  +454.167, Z    +0.000, E1   -22.842, E3 +522158.732}
SPL {X  -162.820, Y  +456.529, Z    +0.000, E1   -22.855, E3 +522170.261}
SPL {X  -162.820, Y  +458.725, Z    +0.000, E1   -22.793, E3 +522181.665}
SPL {X  -162.820, Y  +461.700, Z    +0.000, E1   -22.822, E3 +522196.288}
SPL {X  -162.820, Y  +464.633, Z    +0.000, E1   -22.813, E3 +522210.784}
SPL {X  -162.820, Y  +466.699, Z    +0.000, E1   -22.824, E3 +522220.830}
SPL {X  -162.820, Y  +468.655, Z    +0.000, E1   -22.858, E3 +522230.274}
SPL {X  -162.820, Y  +470.892, Z    +0.000, E1   -22.837, E3 +522241.513}
SPL {X  -162.820, Y  +472.726, Z    +0.000, E1   -22.777, E3 +522251.051}
SPL {X  -162.820, Y  +475.118, Z    +0.000, E1   -22.777, E3 +522263.023}
SPL {X  -162.820, Y  +478.177, Z    +0.000, E1   -22.834, E3 +522277.716}
SPL {X  -162.820, Y  +481.034, Z    +0.000, E1   -22.831, E3 +522291.853}
SPL {X  -162.820, Y  +483.391, Z    +0.000, E1   -22.793, E3 +522303.789}
SPL {X  -162.820, Y  +486.307, Z    +0.000, E1   -22.833, E3 +522318.043}
SPL {X  -162.820, Y  +489.750, Z    +0.000, E1   -22.832, E3 +522335.113}
SPL {X  -162.820, Y  +493.233, Z    +0.000, E1   -22.844, E3 +522352.250}
SPL {X  -162.820, Y  +496.150, Z    +0.000, E1   -22.796, E3 +522366.970}
SPL {X  -162.820, Y  +498.661, Z    +0.000, E1   -22.828, E3 +522379.151}
SPL {X  -162.820, Y  +501.761, Z    +0.000, E1   -22.820, E3 +522394.719}
SPL {X  -162.820, Y  +504.194, Z    +0.000, E1   -22.775, E3 +522406.910}
SPL {X  -162.820, Y  +506.908, Z    +0.000, E1   -22.877, E3 +522419.755}
SPL {X  -162.820, Y  +510.068, Z    +0.000, E1   -22.761, E3 +522436.226}
SPL {X  -162.820, Y  +512.359, Z    +0.000, E1   -22.823, E3 +522446.958}
SPL {X  -162.820, Y  +514.562, Z    +0.000, E1   -22.806, E3 +522458.145}
SPL {X  -162.820, Y  +517.952, Z    +0.000, E1   -22.864, E3 +522474.542}
SPL {X  -162.820, Y  +520.641, Z    +0.000, E1   -22.790, E3 +522488.260}
SPL {X  -162.820, Y  +522.740, Z    +0.000, E1   -22.811, E3 +522498.503}
SPL {X  -162.820, Y  +524.628, Z    +0.000, E1   -22.846, E3 +522507.498}
SPL {X  -162.820, Y  +526.661, Z    +0.000, E1   -22.801, E3 +522518.053}
SPL {X  -162.820, Y  +529.662, Z    +0.000, E1   -22.810, E3 +522532.904}
SPL {X  -162.820, Y  +532.614, Z    +0.000, E1   -22.828, E3 +522547.310}
SPL {X  -162.820, Y  +534.838, Z    +0.000, E1   -22.864, E3 +522557.939}
SPL {X  -162.820, Y  +536.882, Z    +0.000, E1   -22.782, E3 +522568.794}
SPL {X  -162.820, Y  +539.194, Z    +0.000, E1   -22.826, E3 +522579.843}
SPL {X  -162.820, Y  +541.555, Z    +0.000, E1   -22.817, E3 +522591.657}
SPL {X  -162.820, Y  +543.728, Z    +0.000, E1   -22.799, E3 +522602.515}
SPL {X  -162.820, Y  +545.925, Z    +0.000, E1   -22.803, E3 +522613.384}
SPL {X  -162.820, Y  +549.071, Z    +0.000, E1   -22.836, E3 +522628.912}
SPL {X  -162.820, Y  +553.089, Z    +0.000, E1   -22.838, E3 +522648.812}
SPL {X  -162.820, Y  +556.430, Z    +0.000, E1   -22.821, E3 +522665.313}
SPL {X  -162.820, Y  +558.974, Z    +0.000, E1   -22.806, E3 +522678.013}
SPL {X  -162.820, Y  +562.171, Z    +0.000, E1   -22.845, E3 +522693.711}
SPL {X  -162.820, Y  +565.170, Z    +0.000, E1   -22.801, E3 +522708.724}
SPL {X  -162.820, Y  +567.308, Z    +0.000, E1   -22.750, E3 +522719.740}
SPL {X  -162.820, Y  +570.378, Z    +0.000, E1   -22.843, E3 +522734.364}
SPL {X  -162.820, Y  +573.634, Z    +0.000, E1   -22.827, E3 +522750.508}
SPL {X  -162.820, Y  +576.228, Z    +0.000, E1   -22.814, E3 +522763.404}
SPL {X  -162.820, Y  +578.553, Z    +0.000, E1   -22.801, E3 +522775.020}
SPL {X  -162.820, Y  +581.064, Z    +0.000, E1   -22.823, E3 +522787.305}
SPL {X  -162.820, Y  +583.435, Z    +0.000, E1   -22.808, E3 +522799.126}
SPL {X  -162.820, Y  +585.410, Z    +0.000, E1   -22.764, E3 +522809.262}
SPL {X  -162.820, Y  +587.676, Z    +0.000, E1   -22.853, E3 +522819.777}
SPL {X  -162.820, Y  +590.707, Z    +0.000, E1   -22.855, E3 +522834.927}
SPL {X  -162.820, Y  +593.650, Z    +0.000, E1   -22.810, E3 +522849.687}
SPL {X  -162.820, Y  +595.830, Z    +0.000, E1   -22.828, E3 +522860.303}
SPL {X  -162.820, Y  +598.094, Z    +0.000, E1   -22.843, E3 +522871.416}
SPL {X  -162.820, Y  +600.420, Z    +0.000, E1   -22.826, E3 +522883.047}
SPL {X  -162.820, Y  +603.245, Z    +0.000, E1   -22.831, E3 +522897.113}
SPL {X  -162.820, Y  +606.456, Z    +0.000, E1   -22.811, E3 +522913.158}
SPL {X  -162.820, Y  +608.890, Z    +0.000, E1   -22.790, E3 +522925.276}
SPL {X  -162.820, Y  +611.103, Z    +0.000, E1   -22.785, E3 +522936.315}
SPL {X  -162.820, Y  +613.294, Z    +0.000, E1   -22.780, E3 +522947.188}
SPL {X  -162.820, Y  +615.356, Z    +0.000, E1   -22.799, E3 +522957.245}
SPL {X  -162.820, Y  +617.439, Z    +0.000, E1   -22.808, E3 +522967.503}
SPL {X  -162.820, Y  +619.665, Z    +0.000, E1   -22.817, E3 +522978.471}
SPL {X  -162.820, Y  +621.733, Z    +0.000, E1   -22.759, E3 +522989.195}
SPL {X  -162.820, Y  +624.076, Z    +0.000, E1   -22.774, E3 +523000.700}
SPL {X  -162.820, Y  +627.244, Z    +0.000, E1   -22.803, E3 +523016.383}
SPL {X  -162.820, Y  +630.349, Z    +0.000, E1   -22.766, E3 +523031.915}
SPL {X  -162.820, Y  +632.572, Z    +0.000, E1   -22.785, E3 +523042.721}
SPL {X  -162.820, Y  +634.507, Z    +0.000, E1   -22.784, E3 +523052.360}
SPL {X  -162.820, Y  +636.863, Z    +0.000, E1   -22.760, E3 +523064.282}
SPL {X  -162.820, Y  +640.111, Z    +0.000, E1   -22.809, E3 +523080.165}
SPL {X  -162.820, Y  +643.449, Z    +0.000, E1   -22.796, E3 +523096.683}
SPL {X  -162.820, Y  +645.630, Z    +0.000, E1   -22.795, E3 +523107.379}
SPL {X  -162.820, Y  +647.561, Z    +0.000, E1   -22.705, E3 +523117.829}
SPL {X  -162.820, Y  +649.758, Z    +0.000, E1   -22.780, E3 +523128.020}
SPL {X  -162.820, Y  +651.708, Z    +0.000, E1   -22.810, E3 +523137.514}
SPL {X  -162.820, Y  +653.898, Z    +0.000, E1   -22.796, E3 +523148.435}
SPL {X  -162.820, Y  +656.161, Z    +0.000, E1   -22.812, E3 +523159.556}
SPL {X  -162.820, Y  +658.384, Z    +0.000, E1   -22.822, E3 +523170.423}
SPL {X  -162.820, Y  +660.215, Z    +0.000, E1   -22.649, E3 +523181.013}
SPL {X  -162.820, Y  +662.823, Z    +0.000, E1   -22.799, E3 +523192.721}
SPL {X  -162.820, Y  +665.862, Z    +0.000, E1   -22.864, E3 +523207.420}
SPL {X  -162.820, Y  +668.960, Z    +0.000, E1   -22.773, E3 +523223.371}
SPL {X  -162.820, Y  +671.605, Z    +0.000, E1   -22.777, E3 +523236.445}
SPL {X  -162.817, Y  +674.515, Z    +0.000, E1   -22.816, E3 +523250.642}
SPL {X  -162.773, Y  +677.428, Z    +0.000, E1   -22.762, E3 +523265.450}
SPL {X  -162.691, Y  +679.987, Z    +0.000, E1   -22.794, E3 +523277.863}
SPL {X  -162.604, Y  +681.880, Z    +0.000, E1   -22.691, E3 +523288.024}
SPL {X  -162.458, Y  +684.346, Z    +0.000, E1   -22.764, E3 +523299.818}
SPL {X  -162.229, Y  +687.364, Z    +0.000, E1   -22.685, E3 +523315.437}
SPL {X  -161.938, Y  +690.422, Z    +0.000, E1   -22.769, E3 +523329.844}
SPL {X  -161.065, Y  +697.344, Z    +0.000, E1   -25.698, E3 +523338.963}
SPL {X  -158.553, Y  +710.529, Z    +0.000, E1   -30.890, E3 +523352.860}
ENDSPLINE

SPLINE
SPL {X  -161.215, Y  +696.305, Z    +0.000, E1   -20.575, E3 +523379.440}
SPL {X  -161.691, Y  +692.643, Z    +0.000, E1   -17.369, E3 +523395.629}
SPL {X  -162.534, Y  +683.153, Z    +0.000, E1   -10.475, E3 +523421.096}
SPL {X  -162.820, Y  +670.105, Z    +0.000, E1    -2.484, E3 +523413.743}
SPL {X  -162.820, Y  +665.819, Z    +0.000, E1    +0.492, E3 +523416.039}
SPL {X  -162.820, Y  +661.883, Z    +0.000, E1    +3.373, E3 +523420.515}
SPL {X  -162.820, Y  +655.163, Z    +0.000, E1    +8.702, E3 +523420.114}
SPL {X  -162.820, Y  +634.515, Z    +0.000, E1   +26.439, E3 +523412.527}
ENDSPLINE

SPLINE
SPL {X  -162.820, Y  +638.080, Z    +0.000, E1   +18.858, E3 +523442.492}
ENDSPLINE

SPLINE
SPL {X  -162.820, Y  +623.278, Z    +0.000, E1   +28.723, E3 +523444.062}
SPL {X  -162.820, Y  +618.658, Z    +0.000, E1   +26.841, E3 +523472.671}
ENDSPLINE

SPLINE
SPL {X  -162.820, Y  +623.685, Z    +0.000, E1   +22.346, E3 +523484.978}
ENDSPLINE

SPLINE
SPL {X  -162.820, Y  +621.304, Z    +0.000, E1   +22.259, E3 +523497.793}
SPL {X  -162.820, Y  +618.758, Z    +0.000, E1   +22.239, E3 +523510.944}
SPL {X  -162.820, Y  +616.062, Z    +0.000, E1   +22.275, E3 +523524.364}
SPL {X  -162.820, Y  +613.536, Z    +0.000, E1   +22.242, E3 +523537.486}
SPL {X  -162.820, Y  +611.128, Z    +0.000, E1   +22.252, E3 +523549.657}
SPL {X  -162.820, Y  +608.428, Z    +0.000, E1   +22.255, E3 +523563.440}
SPL {X  -162.820, Y  +605.984, Z    +0.000, E1   +22.221, E3 +523576.077}
SPL {X  -162.820, Y  +603.020, Z    +0.000, E1   +22.272, E3 +523590.975}
SPL {X  -162.820, Y  +599.168, Z    +0.000, E1   +22.310, E3 +523610.243}
SPL {X  -162.820, Y  +596.569, Z    +0.000, E1   +22.222, E3 +523623.966}
SPL {X  -162.820, Y  +594.115, Z    +0.000, E1   +22.273, E3 +523636.191}
SPL {X  -162.820, Y  +591.721, Z    +0.000, E1   +22.239, E3 +523648.506}
SPL {X  -162.820, Y  +589.492, Z    +0.000, E1   +22.304, E3 +523659.367}
SPL {X  -162.820, Y  +586.660, Z    +0.000, E1   +22.307, E3 +523673.807}
SPL {X  -162.820, Y  +583.204, Z    +0.000, E1   +22.278, E3 +523691.713}
SPL {X  -162.820, Y  +580.317, Z    +0.000, E1   +22.300, E3 +523705.983}
SPL {X  -162.820, Y  +578.061, Z    +0.000, E1   +22.264, E3 +523717.868}
SPL {X  -162.820, Y  +575.394, Z    +0.000, E1   +22.240, E3 +523731.613}
SPL {X  -162.820, Y  +573.156, Z    +0.000, E1   +22.254, E3 +523742.823}
SPL {X  -162.820, Y  +570.852, Z    +0.000, E1   +22.234, E3 +523754.846}
SPL {X  -162.820, Y  +567.961, Z    +0.000, E1   +22.247, E3 +523769.450}
SPL {X  -162.820, Y  +564.506, Z    +0.000, E1   +22.298, E3 +523786.764}
SPL {X  -162.820, Y  +561.620, Z    +0.000, E1   +22.191, E3 +523802.145}
SPL {X  -162.820, Y  +559.515, Z    +0.000, E1   +22.273, E3 +523812.147}
SPL {X  -162.820, Y  +556.723, Z    +0.000, E1   +22.309, E3 +523826.231}
SPL {X  -162.820, Y  +553.294, Z    +0.000, E1   +22.266, E3 +523844.018}
SPL {X  -162.820, Y  +550.871, Z    +0.000, E1   +22.229, E3 +523856.493}
SPL {X  -162.820, Y  +548.168, Z    +0.000, E1   +22.298, E3 +523869.829}
SPL {X  -162.820, Y  +545.860, Z    +0.000, E1   +22.216, E3 +523882.086}
SPL {X  -162.820, Y  +543.558, Z    +0.000, E1   +22.285, E3 +523893.317}
SPL {X  -162.820, Y  +540.968, Z    +0.000, E1   +22.274, E3 +523906.589}
SPL {X  -162.820, Y  +537.857, Z    +0.000, E1   +22.280, E3 +523922.465}
SPL {X  -162.820, Y  +534.880, Z    +0.000, E1   +22.252, E3 +523937.733}
SPL {X  -162.820, Y  +532.896, Z    +0.000, E1   +22.234, E3 +523947.894}
SPL {X  -162.820, Y  +531.056, Z    +0.000, E1   +22.251, E3 +523957.176}
SPL {X  -162.820, Y  +528.708, Z    +0.000, E1   +22.319, E3 +523968.557}
SPL {X  -162.820, Y  +525.932, Z    +0.000, E1   +22.258, E3 +523983.314}
SPL {X  -162.820, Y  +522.524, Z    +0.000, E1   +22.326, E3 +524000.037}
SPL {X  -162.820, Y  +519.457, Z    +0.000, E1   +22.481, E3 +524014.166}
SPL {X  -162.820, Y  +506.285, Z    +0.000, E1   +28.538, E3 +524025.624}
SPL {X  -162.820, Y  +504.441, Z    +0.000, E1   +27.574, E3 +524039.967}
SPL {X  -162.820, Y  +503.215, Z    +0.000, E1   +26.369, E3 +524053.474}
SPL {X  -162.820, Y  +502.265, Z    +0.000, E1   +25.287, E3 +524065.956}
SPL {X  -162.820, Y  +501.060, Z    +0.000, E1   +24.081, E3 +524080.696}
SPL {X  -162.820, Y  +500.336, Z    +0.000, E1   +23.110, E3 +524091.836}
SPL {X  -162.820, Y  +499.240, Z    +0.000, E1   +22.316, E3 +524104.147}
SPL {X  -162.820, Y  +498.027, Z    +0.000, E1   +21.516, E3 +524117.054}
SPL {X  -162.820, Y  +495.897, Z    +0.000, E1   +21.662, E3 +524126.975}
SPL {X  -162.820, Y  +493.717, Z    +0.000, E1   +21.704, E3 +524138.081}
SPL {X  -162.820, Y  +491.396, Z    +0.000, E1   +21.707, E3 +524150.205}
SPL {X  -162.820, Y  +488.560, Z    +0.000, E1   +21.695, E3 +524165.314}
SPL {X  -162.820, Y  +485.661, Z    +0.000, E1   +21.712, E3 +524180.200}
SPL {X  -162.820, Y  +483.668, Z    +0.000, E1   +21.664, E3 +524191.027}
SPL {X  -162.820, Y  +481.739, Z    +0.000, E1   +21.704, E3 +524200.741}
SPL {X  -162.820, Y  +479.894, Z    +0.000, E1   +21.695, E3 +524210.528}
SPL {X  -162.820, Y  +477.685, Z    +0.000, E1   +21.656, E3 +524222.466}
SPL {X  -162.820, Y  +475.419, Z    +0.000, E1   +21.711, E3 +524233.819}
SPL {X  -162.820, Y  +473.301, Z    +0.000, E1   +21.712, E3 +524244.916}
SPL {X  -162.820, Y  +470.965, Z    +0.000, E1   +21.700, E3 +524257.261}
SPL {X  -162.820, Y  +469.036, Z    +0.000, E1   +21.695, E3 +524267.304}
SPL {X  -162.820, Y  +467.138, Z    +0.000, E1   +21.678, E3 +524277.476}
SPL {X  -162.820, Y  +465.011, Z    +0.000, E1   +21.692, E3 +524288.459}
SPL {X  -162.820, Y  +462.669, Z    +0.000, E1   +21.752, E3 +524300.239}
SPL {X  -162.820, Y  +460.725, Z    +0.000, E1   +21.689, E3 +524310.852}
SPL {X  -162.820, Y  +458.666, Z    +0.000, E1   +21.695, E3 +524321.664}
SPL {X  -162.820, Y  +456.431, Z    +0.000, E1   +21.708, E3 +524333.193}
SPL {X  -162.820, Y  +453.609, Z    +0.000, E1   +21.757, E3 +524347.726}
SPL {X  -162.820, Y  +450.610, Z    +0.000, E1   +21.698, E3 +524363.784}
SPL {X  -162.820, Y  +448.170, Z    +0.000, E1   +21.667, E3 +524376.805}
SPL {X  -162.820, Y  +445.508, Z    +0.000, E1   +21.732, E3 +524390.323}
SPL {X  -162.820, Y  +442.443, Z    +0.000, E1   +21.712, E3 +524406.443}
SPL {X  -162.820, Y  +439.933, Z    +0.000, E1   +21.690, E3 +524419.724}
SPL {X  -162.820, Y  +437.628, Z    +0.000, E1   +21.678, E3 +524431.912}
SPL {X  -162.820, Y  +434.473, Z    +0.000, E1   +21.747, E3 +524448.009}
SPL {X  -162.820, Y  +431.492, Z    +0.000, E1   +21.686, E3 +524463.957}
SPL {X  -162.820, Y  +429.074, Z    +0.000, E1   +21.710, E3 +524476.409}
SPL {X  -162.820, Y  +426.023, Z    +0.000, E1   +21.718, E3 +524492.477}
SPL {X  -162.820, Y  +422.986, Z    +0.000, E1   +21.685, E3 +524508.524}
SPL {X  -162.820, Y  +420.528, Z    +0.000, E1   +21.706, E3 +524521.175}
SPL {X  -162.820, Y  +418.116, Z    +0.000, E1   +21.761, E3 +524533.322}
SPL {X  -162.820, Y  +416.127, Z    +0.000, E1   +21.715, E3 +524544.027}
SPL {X  -162.820, Y  +414.361, Z    +0.000, E1   +21.613, E3 +524554.214}
SPL {X  -162.820, Y  +411.450, Z    +0.000, E1   +21.710, E3 +524568.788}
SPL {X  -162.820, Y  +408.590, Z    +0.000, E1   +21.735, E3 +524583.413}
SPL {X  -162.820, Y  +406.238, Z    +0.000, E1   +21.697, E3 +524596.062}
SPL {X  -162.820, Y  +403.166, Z    +0.000, E1   +21.746, E3 +524611.868}
SPL {X  -162.820, Y  +400.348, Z    +0.000, E1   +21.713, E3 +524626.703}
SPL {X  -162.820, Y  +398.298, Z    +0.000, E1   +21.721, E3 +524637.318}
SPL {X  -162.820, Y  +396.371, Z    +0.000, E1   +21.713, E3 +524647.500}
SPL {X  -162.820, Y  +394.508, Z    +0.000, E1   +21.616, E3 +524658.056}
SPL {X  -162.820, Y  +391.777, Z    +0.000, E1   +21.714, E3 +524671.715}
SPL {X  -162.820, Y  +388.822, Z    +0.000, E1   +21.717, E3 +524687.035}
SPL {X  -162.820, Y  +386.818, Z    +0.000, E1   +21.679, E3 +524697.775}
SPL {X  -162.820, Y  +384.697, Z    +0.000, E1   +21.693, E3 +524708.845}
SPL {X  -162.820, Y  +382.288, Z    +0.000, E1   +21.742, E3 +524720.968}
SPL {X  -162.820, Y  +380.381, Z    +0.000, E1   +21.655, E3 +524731.693}
SPL {X  -162.808, Y  +378.512, Z    +0.000, E1   +21.736, E3 +524740.746}
SPL {X  -162.776, Y  +376.710, Z    +0.000, E1   +21.698, E3 +524750.545}
SPL {X  -162.707, Y  +374.438, Z    +0.000, E1   +21.688, E3 +524762.549}
SPL {X  -162.607, Y  +372.171, Z    +0.000, E1   +21.692, E3 +524774.349}
SPL {X  -162.494, Y  +370.197, Z    +0.000, E1   +21.655, E3 +524784.975}
SPL {X  -162.349, Y  +368.131, Z    +0.000, E1   +21.624, E3 +524796.093}
SPL {X  -162.161, Y  +365.866, Z    +0.000, E1   +21.642, E3 +524807.778}
SPL {X  -161.927, Y  +363.466, Z    +0.000, E1   +21.730, E3 +524819.549}
SPL {X  -160.290, Y  +351.907, Z    +0.000, E1   +27.562, E3 +524827.127}
SPL {X  -159.725, Y  +348.905, Z    +0.000, E1   +26.136, E3 +524852.362}
ENDSPLINE

SPLINE
SPL {X  -160.871, Y  +355.385, Z    +0.000, E1   +21.841, E3 +524861.205}
SPL {X  -161.833, Y  +362.603, Z    +0.000, E1   +17.021, E3 +524871.236}
ENDSPLINE

SPLINE
SPL {X  -160.786, Y  +354.842, Z    +0.000, E1   +19.274, E3 +524903.392}
ENDSPLINE

SPLINE
SPL {X  -162.485, Y  +370.062, Z    +0.000, E1   +10.606, E3 +524909.770}
SPL {X  -162.820, Y  +381.311, Z    +0.000, E1    +4.054, E3 +524900.125}
SPL {X  -162.820, Y  +389.994, Z    +0.000, E1    -2.149, E3 +524894.537}
SPL {X  -162.820, Y  +391.982, Z    +0.000, E1    -3.443, E3 +524904.983}
SPL {X  -162.820, Y  +399.630, Z    +0.000, E1    -9.426, E3 +524907.490}
SPL {X  -162.820, Y  +408.127, Z    +0.000, E1   -18.417, E3 +524893.779}
SPL {X  -162.820, Y  +420.083, Z    +0.000, E1   -24.325, E3 +524914.254}
SPL {X  -162.820, Y  +428.527, Z    +0.000, E1   -26.988, E3 +524931.546}
SPL {X  -162.820, Y  +431.336, Z    +0.000, E1   -24.162, E3 +524961.756}
SPL {X  -162.820, Y  +432.048, Z    +0.000, E1   -22.832, E3 +524976.260}
SPL {X  -162.820, Y  +434.888, Z    +0.000, E1   -22.823, E3 +524990.209}
SPL {X  -162.820, Y  +436.834, Z    +0.000, E1   -22.779, E3 +525000.169}
SPL {X  -162.820, Y  +438.868, Z    +0.000, E1   -22.837, E3 +525009.823}
SPL {X  -162.820, Y  +441.351, Z    +0.000, E1   -22.805, E3 +525022.398}
SPL {X  -162.820, Y  +443.809, Z    +0.000, E1   -22.804, E3 +525034.565}
SPL {X  -162.820, Y  +447.077, Z    +0.000, E1   -22.869, E3 +525050.375}
SPL {X  -162.820, Y  +449.911, Z    +0.000, E1   -22.774, E3 +525064.985}
SPL {X  -162.820, Y  +451.861, Z    +0.000, E1   -22.750, E3 +525074.832}
SPL {X  -162.820, Y  +454.167, Z    +0.000, E1   -22.842, E3 +525085.562}
SPL {X  -162.820, Y  +456.529, Z    +0.000, E1   -22.855, E3 +525097.090}
SPL {X  -162.820, Y  +458.725, Z    +0.000, E1   -22.793, E3 +525108.494}
SPL {X  -162.820, Y  +460.754, Z    +0.000, E1   -22.806, E3 +525118.367}
SPL {X  -162.820, Y  +462.409, Z    +0.000, E1   -22.783, E3 +525126.784}
SPL {X  -162.820, Y  +464.633, Z    +0.000, E1   -22.813, E3 +525137.614}
SPL {X  -162.820, Y  +467.913, Z    +0.000, E1   -22.879, E3 +525153.453}
SPL {X  -162.820, Y  +470.892, Z    +0.000, E1   -22.837, E3 +525168.342}
SPL {X  -162.820, Y  +472.726, Z    +0.000, E1   -22.777, E3 +525177.881}
SPL {X  -162.820, Y  +475.118, Z    +0.000, E1   -22.777, E3 +525189.852}
SPL {X  -162.820, Y  +478.177, Z    +0.000, E1   -22.834, E3 +525204.545}
SPL {X  -162.820, Y  +481.034, Z    +0.000, E1   -22.831, E3 +525218.683}
SPL {X  -162.820, Y  +483.391, Z    +0.000, E1   -22.793, E3 +525230.619}
SPL {X  -162.820, Y  +486.307, Z    +0.000, E1   -22.833, E3 +525244.872}
SPL {X  -162.820, Y  +488.828, Z    +0.000, E1   -22.793, E3 +525257.515}
SPL {X  -162.820, Y  +491.768, Z    +0.000, E1   -22.852, E3 +525271.812}
SPL {X  -162.820, Y  +495.526, Z    +0.000, E1   -22.833, E3 +525290.583}
SPL {X  -162.820, Y  +499.330, Z    +0.000, E1   -22.841, E3 +525309.365}
SPL {X  -162.820, Y  +503.049, Z    +0.000, E1   -22.823, E3 +525327.914}
SPL {X  -162.820, Y  +506.908, Z    +0.000, E1   -22.877, E3 +525346.584}
SPL {X  -162.820, Y  +510.068, Z    +0.000, E1   -22.761, E3 +525363.056}
SPL {X  -162.820, Y  +512.359, Z    +0.000, E1   -22.823, E3 +525373.787}
SPL {X  -162.820, Y  +514.562, Z    +0.000, E1   -22.806, E3 +525384.974}
SPL {X  -162.820, Y  +517.952, Z    +0.000, E1   -22.864, E3 +525401.371}
SPL {X  -162.820, Y  +520.641, Z    +0.000, E1   -22.790, E3 +525415.090}
SPL {X  -162.820, Y  +522.740, Z    +0.000, E1   -22.811, E3 +525425.332}
SPL {X  -162.820, Y  +524.628, Z    +0.000, E1   -22.846, E3 +525434.327}
SPL {X  -162.820, Y  +526.661, Z    +0.000, E1   -22.801, E3 +525444.883}
SPL {X  -162.820, Y  +529.662, Z    +0.000, E1   -22.810, E3 +525459.733}
SPL {X  -162.820, Y  +532.614, Z    +0.000, E1   -22.828, E3 +525474.140}
SPL {X  -162.820, Y  +534.838, Z    +0.000, E1   -22.864, E3 +525484.769}
SPL {X  -162.820, Y  +536.882, Z    +0.000, E1   -22.782, E3 +525495.623}
SPL {X  -162.820, Y  +539.194, Z    +0.000, E1   -22.826, E3 +525506.672}
SPL {X  -162.820, Y  +541.555, Z    +0.000, E1   -22.817, E3 +525518.486}
SPL {X  -162.820, Y  +543.728, Z    +0.000, E1   -22.799, E3 +525529.344}
SPL {X  -162.820, Y  +545.925, Z    +0.000, E1   -22.803, E3 +525540.214}
SPL {X  -162.820, Y  +548.328, Z    +0.000, E1   -22.796, E3 +525552.209}
SPL {X  -162.820, Y  +551.027, Z    +0.000, E1   -22.819, E3 +525565.402}
SPL {X  -162.820, Y  +553.721, Z    +0.000, E1   -22.807, E3 +525578.846}
SPL {X  -162.820, Y  +556.430, Z    +0.000, E1   -22.821, E3 +525592.142}
SPL {X  -162.820, Y  +559.675, Z    +0.000, E1   -22.837, E3 +525608.222}
SPL {X  -162.820, Y  +562.799, Z    +0.000, E1   -22.814, E3 +525623.729}
SPL {X  -162.820, Y  +565.170, Z    +0.000, E1   -22.801, E3 +525635.554}
SPL {X  -162.820, Y  +568.020, Z    +0.000, E1   -22.787, E3 +525649.940}
SPL {X  -162.820, Y  +570.992, Z    +0.000, E1   -22.834, E3 +525664.159}
SPL {X  -162.820, Y  +572.901, Z    +0.000, E1   -22.775, E3 +525674.028}
SPL {X  -162.820, Y  +575.638, Z    +0.000, E1   -22.855, E3 +525687.137}
SPL {X  -162.820, Y  +578.553, Z    +0.000, E1   -22.801, E3 +525701.850}
SPL {X  -162.820, Y  +581.064, Z    +0.000, E1   -22.823, E3 +525714.134}
SPL {X  -162.820, Y  +583.435, Z    +0.000, E1   -22.808, E3 +525725.956}
SPL {X  -162.820, Y  +585.410, Z    +0.000, E1   -22.764, E3 +525736.091}
SPL {X  -162.820, Y  +587.676, Z    +0.000, E1   -22.853, E3 +525746.606}
SPL {X  -162.820, Y  +589.682, Z    +0.000, E1   -22.776, E3 +525757.136}
SPL {X  -162.820, Y  +591.720, Z    +0.000, E1   -22.868, E3 +525766.447}
SPL {X  -162.820, Y  +593.650, Z    +0.000, E1   -22.810, E3 +525776.517}
SPL {X  -162.820, Y  +595.830, Z    +0.000, E1   -22.828, E3 +525787.132}
SPL {X  -162.820, Y  +598.094, Z    +0.000, E1   -22.843, E3 +525798.246}
SPL {X  -162.820, Y  +600.420, Z    +0.000, E1   -22.826, E3 +525809.877}
SPL {X  -162.820, Y  +602.573, Z    +0.000, E1   -22.830, E3 +525820.462}
SPL {X  -162.820, Y  +604.828, Z    +0.000, E1   -22.784, E3 +525832.100}
SPL {X  -162.820, Y  +608.133, Z    +0.000, E1   -22.831, E3 +525848.218}
SPL {X  -162.820, Y  +611.103, Z    +0.000, E1   -22.785, E3 +525863.144}
SPL {X  -162.820, Y  +613.294, Z    +0.000, E1   -22.780, E3 +525874.017}
SPL {X  -162.820, Y  +615.356, Z    +0.000, E1   -22.799, E3 +525884.074}
SPL {X  -162.820, Y  +617.439, Z    +0.000, E1   -22.808, E3 +525894.332}
SPL {X  -162.820, Y  +619.665, Z    +0.000, E1   -22.817, E3 +525905.300}
SPL {X  -162.820, Y  +621.733, Z    +0.000, E1   -22.759, E3 +525916.025}
SPL {X  -162.820, Y  +624.076, Z    +0.000, E1   -22.774, E3 +525927.530}
SPL {X  -162.820, Y  +626.527, Z    +0.000, E1   -22.768, E3 +525939.772}
SPL {X  -162.820, Y  +629.758, Z    +0.000, E1   -22.800, E3 +525955.701}
SPL {X  -162.820, Y  +632.572, Z    +0.000, E1   -22.785, E3 +525969.550}
SPL {X  -162.820, Y  +634.507, Z    +0.000, E1   -22.784, E3 +525979.189}
SPL {X  -162.820, Y  +636.863, Z    +0.000, E1   -22.760, E3 +525991.111}
SPL {X  -162.820, Y  +640.111, Z    +0.000, E1   -22.809, E3 +526006.994}
SPL {X  -162.820, Y  +643.449, Z    +0.000, E1   -22.796, E3 +526023.512}
SPL {X  -162.820, Y  +645.630, Z    +0.000, E1   -22.795, E3 +526034.208}
SPL {X  -162.820, Y  +647.561, Z    +0.000, E1   -22.705, E3 +526044.659}
SPL {X  -162.820, Y  +649.758, Z    +0.000, E1   -22.780, E3 +526054.849}
SPL {X  -162.820, Y  +651.708, Z    +0.000, E1   -22.810, E3 +526064.343}
SPL {X  -162.820, Y  +653.898, Z    +0.000, E1   -22.796, E3 +526075.264}
SPL {X  -162.820, Y  +656.161, Z    +0.000, E1   -22.812, E3 +526086.386}
SPL {X  -162.820, Y  +658.384, Z    +0.000, E1   -22.822, E3 +526097.252}
SPL {X  -162.820, Y  +660.215, Z    +0.000, E1   -22.649, E3 +526107.842}
SPL {X  -162.820, Y  +662.823, Z    +0.000, E1   -22.799, E3 +526119.550}
SPL {X  -162.820, Y  +665.112, Z    +0.000, E1   -22.835, E3 +526130.605}
SPL {X  -162.820, Y  +667.016, Z    +0.000, E1   -22.823, E3 +526140.033}
SPL {X  -162.820, Y  +668.960, Z    +0.000, E1   -22.773, E3 +526150.201}
SPL {X  -162.820, Y  +672.333, Z    +0.000, E1   -22.837, E3 +526166.537}
SPL {X  -162.812, Y  +675.071, Z    +0.000, E1   -22.742, E3 +526180.682}
SPL {X  -162.773, Y  +677.428, Z    +0.000, E1   -22.762, E3 +526192.279}
SPL {X  -162.691, Y  +679.987, Z    +0.000, E1   -22.794, E3 +526204.693}
SPL {X  -162.604, Y  +681.880, Z    +0.000, E1   -22.691, E3 +526214.853}
SPL {X  -162.458, Y  +684.346, Z    +0.000, E1   -22.764, E3 +526226.647}
SPL {X  -162.296, Y  +686.547, Z    +0.000, E1   -22.660, E3 +526238.264}
SPL {X  -162.164, Y  +688.106, Z    +0.000, E1   -22.661, E3 +526245.997}
SPL {X  -161.938, Y  +690.422, Z    +0.000, E1   -22.769, E3 +526256.673}
SPL {X  -161.065, Y  +697.344, Z    +0.000, E1   -25.698, E3 +526265.792}
SPL {X  -158.730, Y  +709.763, Z    +0.000, E1   -31.225, E3 +526274.466}
ENDSPLINE

SPLINE
SPL {X  -160.932, Y  +698.225, Z    +0.000, E1   -21.712, E3 +526305.575}
SPL {X  -161.917, Y  +690.622, Z    +0.000, E1   -16.445, E3 +526319.176}
ENDSPLINE

SPLINE
SPL {X  -161.349, Y  +695.340, Z    +0.000, E1   -18.625, E3 +526326.794}
ENDSPLINE

SPLINE
SPL {X  -162.534, Y  +683.153, Z    +0.000, E1   -10.475, E3 +526347.925}
SPL {X  -162.820, Y  +667.630, Z    +0.000, E1    -0.882, E3 +526341.901}
SPL {X  -162.820, Y  +661.883, Z    +0.000, E1    +3.373, E3 +526347.344}
SPL {X  -162.820, Y  +655.163, Z    +0.000, E1    +8.702, E3 +526346.943}
SPL {X  -162.820, Y  +634.515, Z    +0.000, E1   +26.439, E3 +526339.356}
ENDSPLINE

SPLINE
SPL {X  -162.820, Y  +638.080, Z    +0.000, E1   +18.858, E3 +526369.321}
ENDSPLINE

SPLINE
SPL {X  -162.820, Y  +623.278, Z    +0.000, E1   +28.723, E3 +526370.892}
SPL {X  -162.820, Y  +618.658, Z    +0.000, E1   +26.841, E3 +526399.500}
ENDSPLINE

SPLINE
SPL {X  -162.820, Y  +623.685, Z    +0.000, E1   +22.346, E3 +526411.807}
ENDSPLINE

SPLINE
SPL {X  -162.820, Y  +621.304, Z    +0.000, E1   +22.259, E3 +526424.622}
SPL {X  -162.820, Y  +618.758, Z    +0.000, E1   +22.239, E3 +526437.773}
SPL {X  -162.820, Y  +616.062, Z    +0.000, E1   +22.275, E3 +526451.194}
SPL {X  -162.820, Y  +613.536, Z    +0.000, E1   +22.242, E3 +526464.315}
SPL {X  -162.820, Y  +610.461, Z    +0.000, E1   +22.264, E3 +526479.946}
SPL {X  -162.820, Y  +607.796, Z    +0.000, E1   +22.261, E3 +526493.318}
SPL {X  -162.820, Y  +605.178, Z    +0.000, E1   +22.267, E3 +526506.801}
SPL {X  -162.820, Y  +602.350, Z    +0.000, E1   +22.224, E3 +526521.419}
SPL {X  -162.820, Y  +599.842, Z    +0.000, E1   +22.298, E3 +526533.570}
SPL {X  -162.820, Y  +597.194, Z    +0.000, E1   +22.253, E3 +526547.491}
SPL {X  -162.820, Y  +594.115, Z    +0.000, E1   +22.273, E3 +526563.020}
SPL {X  -162.820, Y  +591.721, Z    +0.000, E1   +22.239, E3 +526575.335}
SPL {X  -162.820, Y  +589.492, Z    +0.000, E1   +22.304, E3 +526586.196}
SPL {X  -162.820, Y  +587.447, Z    +0.000, E1   +22.279, E3 +526596.725}
SPL {X  -162.820, Y  +585.192, Z    +0.000, E1   +22.298, E3 +526608.135}
SPL {X  -162.820, Y  +582.610, Z    +0.000, E1   +22.234, E3 +526621.759}
SPL {X  -162.820, Y  +580.317, Z    +0.000, E1   +22.300, E3 +526632.812}
SPL {X  -162.820, Y  +578.878, Z    +0.000, E1   +22.272, E3 +526640.322}
SPL {X  -162.820, Y  +576.856, Z    +0.000, E1   +22.233, E3 +526651.080}
SPL {X  -162.820, Y  +574.811, Z    +0.000, E1   +22.236, E3 +526661.344}
SPL {X  -162.820, Y  +572.645, Z    +0.000, E1   +22.246, E3 +526672.439}
SPL {X  -162.820, Y  +569.475, Z    +0.000, E1   +22.269, E3 +526688.445}
SPL {X  -162.820, Y  +565.838, Z    +0.000, E1   +22.271, E3 +526707.040}
SPL {X  -162.820, Y  +562.162, Z    +0.000, E1   +22.252, E3 +526725.857}
SPL {X  -162.820, Y  +559.515, Z    +0.000, E1   +22.273, E3 +526738.976}
SPL {X  -162.820, Y  +556.723, Z    +0.000, E1   +22.309, E3 +526753.060}
SPL {X  -162.820, Y  +553.294, Z    +0.000, E1   +22.266, E3 +526770.848}
SPL {X  -162.820, Y  +550.136, Z    +0.000, E1   +22.258, E3 +526786.961}
SPL {X  -162.820, Y  +546.694, Z    +0.000, E1   +22.290, E3 +526804.283}
SPL {X  -162.820, Y  +543.558, Z    +0.000, E1   +22.285, E3 +526820.146}
SPL {X  -162.820, Y  +541.633, Z    +0.000, E1   +22.257, E3 +526830.074}
SPL {X  -162.820, Y  +539.116, Z    +0.000, E1   +22.302, E3 +526842.685}
SPL {X  -162.820, Y  +535.523, Z    +0.000, E1   +22.266, E3 +526861.347}
SPL {X  -162.820, Y  +531.757, Z    +0.000, E1   +22.276, E3 +526880.401}
SPL {X  -162.820, Y  +527.980, Z    +0.000, E1   +22.326, E3 +526899.232}
SPL {X  -162.820, Y  +524.599, Z    +0.000, E1   +22.287, E3 +526916.629}
SPL {X  -162.820, Y  +522.011, Z    +0.000, E1   +22.282, E3 +526929.706}
SPL {X  -162.820, Y  +519.457, Z    +0.000, E1   +22.481, E3 +526940.996}
SPL {X  -162.820, Y  +505.859, Z    +0.000, E1   +28.367, E3 +526955.479}
SPL {X  -162.820, Y  +504.131, Z    +0.000, E1   +27.325, E3 +526969.617}
SPL {X  -162.820, Y  +503.215, Z    +0.000, E1   +26.369, E3 +526980.303}
SPL {X  -162.820, Y  +502.265, Z    +0.000, E1   +25.287, E3 +526992.785}
SPL {X  -162.820, Y  +501.060, Z    +0.000, E1   +24.081, E3 +527007.525}
SPL {X  -162.820, Y  +500.336, Z    +0.000, E1   +23.110, E3 +527018.665}
SPL {X  -162.820, Y  +499.240, Z    +0.000, E1   +22.316, E3 +527030.976}
SPL {X  -162.820, Y  +498.027, Z    +0.000, E1   +21.516, E3 +527043.884}
SPL {X  -162.820, Y  +495.897, Z    +0.000, E1   +21.662, E3 +527053.804}
SPL {X  -162.820, Y  +493.717, Z    +0.000, E1   +21.704, E3 +527064.910}
SPL {X  -162.820, Y  +491.396, Z    +0.000, E1   +21.707, E3 +527077.034}
SPL {X  -162.820, Y  +488.560, Z    +0.000, E1   +21.695, E3 +527092.144}
SPL {X  -162.820, Y  +485.661, Z    +0.000, E1   +21.712, E3 +527107.029}
SPL {X  -162.820, Y  +483.668, Z    +0.000, E1   +21.664, E3 +527117.856}
SPL {X  -162.820, Y  +481.739, Z    +0.000, E1   +21.704, E3 +527127.570}
SPL {X  -162.820, Y  +479.894, Z    +0.000, E1   +21.695, E3 +527137.358}
SPL {X  -162.820, Y  +477.685, Z    +0.000, E1   +21.656, E3 +527149.295}
SPL {X  -162.820, Y  +475.419, Z    +0.000, E1   +21.711, E3 +527160.648}
SPL {X  -162.820, Y  +473.301, Z    +0.000, E1   +21.712, E3 +527171.745}
SPL {X  -162.820, Y  +470.965, Z    +0.000, E1   +21.700, E3 +527184.090}
SPL {X  -162.820, Y  +469.036, Z    +0.000, E1   +21.695, E3 +527194.134}
SPL {X  -162.820, Y  +467.138, Z    +0.000, E1   +21.678, E3 +527204.305}
SPL {X  -162.820, Y  +465.011, Z    +0.000, E1   +21.692, E3 +527215.288}
SPL {X  -162.820, Y  +462.669, Z    +0.000, E1   +21.752, E3 +527227.068}
SPL {X  -162.820, Y  +460.725, Z    +0.000, E1   +21.689, E3 +527237.681}
SPL {X  -162.820, Y  +458.666, Z    +0.000, E1   +21.695, E3 +527248.493}
SPL {X  -162.820, Y  +456.431, Z    +0.000, E1   +21.708, E3 +527260.022}
SPL {X  -162.820, Y  +453.609, Z    +0.000, E1   +21.757, E3 +527274.556}
SPL {X  -162.820, Y  +450.610, Z    +0.000, E1   +21.698, E3 +527290.613}
SPL {X  -162.820, Y  +448.170, Z    +0.000, E1   +21.667, E3 +527303.634}
SPL {X  -162.820, Y  +446.246, Z    +0.000, E1   +21.696, E3 +527313.452}
SPL {X  -162.820, Y  +443.784, Z    +0.000, E1   +21.713, E3 +527326.238}
SPL {X  -162.820, Y  +441.754, Z    +0.000, E1   +21.708, E3 +527336.790}
SPL {X  -162.820, Y  +439.933, Z    +0.000, E1   +21.690, E3 +527346.554}
SPL {X  -162.820, Y  +437.628, Z    +0.000, E1   +21.678, E3 +527358.742}
SPL {X  -162.820, Y  +435.262, Z    +0.000, E1   +21.727, E3 +527370.677}
SPL {X  -162.820, Y  +433.510, Z    +0.000, E1   +21.692, E3 +527380.091}
SPL {X  -162.820, Y  +431.492, Z    +0.000, E1   +21.686, E3 +527390.786}
SPL {X  -162.820, Y  +429.074, Z    +0.000, E1   +21.710, E3 +527403.238}
SPL {X  -162.820, Y  +427.020, Z    +0.000, E1   +21.674, E3 +527414.240}
SPL {X  -162.820, Y  +424.525, Z    +0.000, E1   +21.712, E3 +527427.153}
SPL {X  -162.820, Y  +421.144, Z    +0.000, E1   +21.719, E3 +527444.820}
SPL {X  -162.820, Y  +418.116, Z    +0.000, E1   +21.761, E3 +527460.151}
SPL {X  -162.820, Y  +416.127, Z    +0.000, E1   +21.715, E3 +527470.856}
SPL {X  -162.820, Y  +414.361, Z    +0.000, E1   +21.613, E3 +527481.043}
SPL {X  -162.820, Y  +412.134, Z    +0.000, E1   +21.697, E3 +527491.988}
SPL {X  -162.820, Y  +409.248, Z    +0.000, E1   +21.741, E3 +527506.923}
SPL {X  -162.820, Y  +406.238, Z    +0.000, E1   +21.697, E3 +527522.891}
SPL {X  -162.820, Y  +404.001, Z    +0.000, E1   +21.723, E3 +527534.321}
SPL {X  -162.820, Y  +402.223, Z    +0.000, E1   +21.697, E3 +527543.806}
SPL {X  -162.820, Y  +400.348, Z    +0.000, E1   +21.713, E3 +527553.532}
SPL {X  -162.820, Y  +398.298, Z    +0.000, E1   +21.721, E3 +527564.148}
SPL {X  -162.820, Y  +396.371, Z    +0.000, E1   +21.713, E3 +527574.329}
SPL {X  -162.820, Y  +394.508, Z    +0.000, E1   +21.616, E3 +527584.885}
SPL {X  -162.820, Y  +391.777, Z    +0.000, E1   +21.714, E3 +527598.544}
SPL {X  -162.820, Y  +388.822, Z    +0.000, E1   +21.717, E3 +527613.864}
SPL {X  -162.820, Y  +386.818, Z    +0.000, E1   +21.679, E3 +527624.604}
SPL {X  -162.820, Y  +384.697, Z    +0.000, E1   +21.693, E3 +527635.674}
SPL {X  -162.820, Y  +382.288, Z    +0.000, E1   +21.742, E3 +527647.798}
SPL {X  -162.817, Y  +379.520, Z    +0.000, E1   +21.723, E3 +527662.635}
SPL {X  -162.776, Y  +376.710, Z    +0.000, E1   +21.698, E3 +527677.374}
SPL {X  -162.707, Y  +374.438, Z    +0.000, E1   +21.688, E3 +527689.378}
SPL {X  -162.607, Y  +372.171, Z    +0.000, E1   +21.692, E3 +527701.178}
SPL {X  -162.494, Y  +370.197, Z    +0.000, E1   +21.655, E3 +527711.804}
SPL {X  -162.349, Y  +368.131, Z    +0.000, E1   +21.624, E3 +527722.922}
SPL {X  -162.161, Y  +365.866, Z    +0.000, E1   +21.642, E3 +527734.607}
SPL {X  -161.927, Y  +363.466, Z    +0.000, E1   +21.730, E3 +527746.379}
SPL {X  -160.290, Y  +351.907, Z    +0.000, E1   +27.562, E3 +527753.956}
SPL {X  -159.725, Y  +348.905, Z    +0.000, E1   +26.136, E3 +527779.192}
ENDSPLINE

SPLINE
SPL {X  -160.871, Y  +355.385, Z    +0.000, E1   +21.841, E3 +527788.035}
SPL {X  -161.833, Y  +362.603, Z    +0.000, E1   +17.021, E3 +527798.066}
ENDSPLINE

SPLINE
SPL {X  -160.786, Y  +354.842, Z    +0.000, E1   +19.274, E3 +527830.221}
ENDSPLINE

SPLINE
SPL {X  -162.485, Y  +370.062, Z    +0.000, E1   +10.606, E3 +527836.599}
SPL {X  -162.820, Y  +381.311, Z    +0.000, E1    +4.054, E3 +527826.954}
SPL {X  -162.820, Y  +389.994, Z    +0.000, E1    -2.149, E3 +527821.367}
SPL {X  -162.820, Y  +391.982, Z    +0.000, E1    -3.443, E3 +527831.812}
SPL {X  -162.820, Y  +399.630, Z    +0.000, E1    -9.426, E3 +527834.319}
SPL {X  -162.820, Y  +408.127, Z    +0.000, E1   -18.417, E3 +527820.608}
SPL {X  -162.820, Y  +420.083, Z    +0.000, E1   -24.325, E3 +527841.083}
SPL {X  -162.820, Y  +428.527, Z    +0.000, E1   -26.988, E3 +527858.375}
SPL {X  -162.820, Y  +431.336, Z    +0.000, E1   -24.162, E3 +527888.585}
SPL {X  -162.820, Y  +432.048, Z    +0.000, E1   -22.832, E3 +527903.089}
SPL {X  -162.820, Y  +434.888, Z    +0.000, E1   -22.823, E3 +527917.039}
SPL {X  -162.820, Y  +436.834, Z    +0.000, E1   -22.779, E3 +527926.999}
SPL {X  -162.820, Y  +438.868, Z    +0.000, E1   -22.837, E3 +527936.652}
SPL {X  -162.820, Y  +441.351, Z    +0.000, E1   -22.805, E3 +527949.228}
SPL {X  -162.820, Y  +443.809, Z    +0.000, E1   -22.804, E3 +527961.394}
SPL {X  -162.820, Y  +447.077, Z    +0.000, E1   -22.869, E3 +527977.204}
SPL {X  -162.820, Y  +449.911, Z    +0.000, E1   -22.774, E3 +527991.814}
SPL {X  -162.820, Y  +451.861, Z    +0.000, E1   -22.750, E3 +528001.661}
SPL {X  -162.820, Y  +454.167, Z    +0.000, E1   -22.842, E3 +528012.391}
SPL {X  -162.820, Y  +456.529, Z    +0.000, E1   -22.855, E3 +528023.919}
SPL {X  -162.820, Y  +458.725, Z    +0.000, E1   -22.793, E3 +528035.324}
SPL {X  -162.820, Y  +460.754, Z    +0.000, E1   -22.806, E3 +528045.197}
SPL {X  -162.820, Y  +462.409, Z    +0.000, E1   -22.783, E3 +528053.613}
SPL {X  -162.820, Y  +464.633, Z    +0.000, E1   -22.813, E3 +528064.443}
SPL {X  -162.820, Y  +467.913, Z    +0.000, E1   -22.879, E3 +528080.282}
SPL {X  -162.820, Y  +470.892, Z    +0.000, E1   -22.837, E3 +528095.171}
SPL {X  -162.820, Y  +472.726, Z    +0.000, E1   -22.777, E3 +528104.710}
SPL {X  -162.820, Y  +475.118, Z    +0.000, E1   -22.777, E3 +528116.681}
SPL {X  -162.820, Y  +477.389, Z    +0.000, E1   -22.803, E3 +528127.598}
SPL {X  -162.820, Y  +478.914, Z    +0.000, E1   -22.821, E3 +528134.990}
SPL {X  -162.820, Y  +481.034, Z    +0.000, E1   -22.831, E3 +528145.512}
SPL {X  -162.820, Y  +484.256, Z    +0.000, E1   -22.840, E3 +528161.530}
SPL {X  -162.820, Y  +487.952, Z    +0.000, E1   -22.824, E3 +528179.961}
SPL {X  -162.820, Y  +490.653, Z    +0.000, E1   -22.810, E3 +528193.231}
SPL {X  -162.820, Y  +493.233, Z    +0.000, E1   -22.844, E3 +528205.908}
SPL {X  -162.820, Y  +496.150, Z    +0.000, E1   -22.796, E3 +528220.628}
SPL {X  -162.820, Y  +498.661, Z    +0.000, E1   -22.828, E3 +528232.809}
SPL {X  -162.820, Y  +501.761, Z    +0.000, E1   -22.820, E3 +528248.378}
SPL {X  -162.820, Y  +505.323, Z    +0.000, E1   -22.838, E3 +528265.824}
SPL {X  -162.820, Y  +507.875, Z    +0.000, E1   -22.849, E3 +528278.192}
SPL {X  -162.820, Y  +510.068, Z    +0.000, E1   -22.761, E3 +528289.885}
SPL {X  -162.820, Y  +512.359, Z    +0.000, E1   -22.823, E3 +528300.616}
SPL {X  -162.820, Y  +514.562, Z    +0.000, E1   -22.806, E3 +528311.803}
SPL {X  -162.820, Y  +517.952, Z    +0.000, E1   -22.864, E3 +528328.201}
SPL {X  -162.820, Y  +520.641, Z    +0.000, E1   -22.790, E3 +528341.919}
SPL {X  -162.820, Y  +522.740, Z    +0.000, E1   -22.811, E3 +528352.162}
SPL {X  -162.820, Y  +524.628, Z    +0.000, E1   -22.846, E3 +528361.157}
SPL {X  -162.820, Y  +526.661, Z    +0.000, E1   -22.801, E3 +528371.712}
SPL {X  -162.820, Y  +529.662, Z    +0.000, E1   -22.810, E3 +528386.563}
SPL {X  -162.820, Y  +532.614, Z    +0.000, E1   -22.828, E3 +528400.969}
SPL {X  -162.820, Y  +534.838, Z    +0.000, E1   -22.864, E3 +528411.598}
SPL {X  -162.820, Y  +536.882, Z    +0.000, E1   -22.782, E3 +528422.453}
SPL {X  -162.820, Y  +539.194, Z    +0.000, E1   -22.826, E3 +528433.501}
SPL {X  -162.820, Y  +541.555, Z    +0.000, E1   -22.817, E3 +528445.316}
SPL {X  -162.820, Y  +543.728, Z    +0.000, E1   -22.799, E3 +528456.173}
SPL {X  -162.820, Y  +545.925, Z    +0.000, E1   -22.803, E3 +528467.043}
SPL {X  -162.820, Y  +548.328, Z    +0.000, E1   -22.796, E3 +528479.039}
SPL {X  -162.820, Y  +551.027, Z    +0.000, E1   -22.819, E3 +528492.231}
SPL {X  -162.820, Y  +553.721, Z    +0.000, E1   -22.807, E3 +528505.676}
SPL {X  -162.820, Y  +556.430, Z    +0.000, E1   -22.821, E3 +528518.972}
SPL {X  -162.820, Y  +559.675, Z    +0.000, E1   -22.837, E3 +528535.052}
SPL {X  -162.820, Y  +562.799, Z    +0.000, E1   -22.814, E3 +528550.558}
SPL {X  -162.820, Y  +565.170, Z    +0.000, E1   -22.801, E3 +528562.383}
SPL {X  -162.820, Y  +568.020, Z    +0.000, E1   -22.787, E3 +528576.769}
SPL {X  -162.820, Y  +570.992, Z    +0.000, E1   -22.834, E3 +528590.989}
SPL {X  -162.820, Y  +572.901, Z    +0.000, E1   -22.775, E3 +528600.857}
SPL {X  -162.820, Y  +575.638, Z    +0.000, E1   -22.855, E3 +528613.967}
SPL {X  -162.820, Y  +578.553, Z    +0.000, E1   -22.801, E3 +528628.679}
SPL {X  -162.820, Y  +581.064, Z    +0.000, E1   -22.823, E3 +528640.963}
SPL {X  -162.820, Y  +583.435, Z    +0.000, E1   -22.808, E3 +528652.785}
SPL {X  -162.820, Y  +585.410, Z    +0.000, E1   -22.764, E3 +528662.921}
SPL {X  -162.820, Y  +587.676, Z    +0.000, E1   -22.853, E3 +528673.435}
SPL {X  -162.820, Y  +589.682, Z    +0.000, E1   -22.776, E3 +528683.965}
SPL {X  -162.820, Y  +591.720, Z    +0.000, E1   -22.868, E3 +528693.276}
SPL {X  -162.820, Y  +593.650, Z    +0.000, E1   -22.810, E3 +528703.346}
SPL {X  -162.820, Y  +595.830, Z    +0.000, E1   -22.828, E3 +528713.962}
SPL {X  -162.820, Y  +598.094, Z    +0.000, E1   -22.843, E3 +528725.075}
SPL {X  -162.820, Y  +600.420, Z    +0.000, E1   -22.826, E3 +528736.706}
SPL {X  -162.820, Y  +602.573, Z    +0.000, E1   -22.830, E3 +528747.291}
SPL {X  -162.820, Y  +604.828, Z    +0.000, E1   -22.784, E3 +528758.930}
SPL {X  -162.820, Y  +608.133, Z    +0.000, E1   -22.831, E3 +528775.047}
SPL {X  -162.820, Y  +611.103, Z    +0.000, E1   -22.785, E3 +528789.973}
SPL {X  -162.820, Y  +613.294, Z    +0.000, E1   -22.780, E3 +528800.846}
SPL {X  -162.820, Y  +615.356, Z    +0.000, E1   -22.799, E3 +528810.903}
SPL {X  -162.820, Y  +617.439, Z    +0.000, E1   -22.808, E3 +528821.162}
SPL {X  -162.820, Y  +619.665, Z    +0.000, E1   -22.817, E3 +528832.130}
SPL {X  -162.820, Y  +621.733, Z    +0.000, E1   -22.759, E3 +528842.854}
SPL {X  -162.820, Y  +624.076, Z    +0.000, E1   -22.774, E3 +528854.359}
SPL {X  -162.820, Y  +627.244, Z    +0.000, E1   -22.803, E3 +528870.041}
SPL {X  -162.820, Y  +630.349, Z    +0.000, E1   -22.766, E3 +528885.573}
SPL {X  -162.820, Y  +632.572, Z    +0.000, E1   -22.785, E3 +528896.380}
SPL {X  -162.820, Y  +634.507, Z    +0.000, E1   -22.784, E3 +528906.019}
SPL {X  -162.820, Y  +636.863, Z    +0.000, E1   -22.760, E3 +528917.941}
SPL {X  -162.820, Y  +640.111, Z    +0.000, E1   -22.809, E3 +528933.823}
SPL {X  -162.820, Y  +643.449, Z    +0.000, E1   -22.796, E3 +528950.341}
SPL {X  -162.820, Y  +645.630, Z    +0.000, E1   -22.795, E3 +528961.037}
SPL {X  -162.820, Y  +647.561, Z    +0.000, E1   -22.705, E3 +528971.488}
SPL {X  -162.820, Y  +649.758, Z    +0.000, E1   -22.780, E3 +528981.678}
SPL {X  -162.820, Y  +651.708, Z    +0.000, E1   -22.810, E3 +528991.173}
SPL {X  -162.820, Y  +653.898, Z    +0.000, E1   -22.796, E3 +529002.093}
SPL {X  -162.820, Y  +656.161, Z    +0.000, E1   -22.812, E3 +529013.215}
SPL {X  -162.820, Y  +658.384, Z    +0.000, E1   -22.822, E3 +529024.081}
SPL {X  -162.820, Y  +660.215, Z    +0.000, E1   -22.649, E3 +529034.672}
SPL {X  -162.820, Y  +662.823, Z    +0.000, E1   -22.799, E3 +529046.380}
SPL {X  -162.820, Y  +665.862, Z    +0.000, E1   -22.864, E3 +529061.079}
SPL {X  -162.820, Y  +668.960, Z    +0.000, E1   -22.773, E3 +529077.030}
SPL {X  -162.820, Y  +671.605, Z    +0.000, E1   -22.777, E3 +529090.104}
SPL {X  -162.817, Y  +674.515, Z    +0.000, E1   -22.816, E3 +529104.301}
SPL {X  -162.773, Y  +677.428, Z    +0.000, E1   -22.762, E3 +529119.108}
SPL {X  -162.691, Y  +679.987, Z    +0.000, E1   -22.794, E3 +529131.522}
SPL {X  -162.559, Y  +682.717, Z    +0.000, E1   -22.726, E3 +529145.705}
SPL {X  -162.404, Y  +685.137, Z    +0.000, E1   -22.766, E3 +529157.228}
SPL {X  -162.229, Y  +687.364, Z    +0.000, E1   -22.685, E3 +529169.096}
SPL {X  -161.938, Y  +690.422, Z    +0.000, E1   -22.769, E3 +529183.502}
SPL {X  -161.065, Y  +697.344, Z    +0.000, E1   -25.698, E3 +529192.622}
SPL {X  -158.730, Y  +709.763, Z    +0.000, E1   -31.225, E3 +529201.295}
ENDSPLINE

SPLINE
SPL {X  -160.932, Y  +698.225, Z    +0.000, E1   -21.712, E3 +529232.404}
SPL {X  -161.691, Y  +692.643, Z    +0.000, E1   -17.369, E3 +529249.287}
SPL {X  -162.534, Y  +683.153, Z    +0.000, E1   -10.475, E3 +529274.754}
SPL {X  -162.820, Y  +667.630, Z    +0.000, E1    -0.882, E3 +529268.731}
SPL {X  -162.820, Y  +661.883, Z    +0.000, E1    +3.373, E3 +529274.174}
SPL {X  -162.820, Y  +655.163, Z    +0.000, E1    +8.702, E3 +529273.772}
SPL {X  -162.820, Y  +634.515, Z    +0.000, E1   +26.439, E3 +529266.186}
ENDSPLINE

SPLINE
SPL {X  -162.820, Y  +638.080, Z    +0.000, E1   +18.858, E3 +529296.150}
ENDSPLINE

SPLINE
SPL {X  -162.820, Y  +623.278, Z    +0.000, E1   +28.723, E3 +529297.721}
SPL {X  -162.820, Y  +618.658, Z    +0.000, E1   +26.841, E3 +529326.330}
ENDSPLINE

SPLINE
SPL {X  -162.820, Y  +623.685, Z    +0.000, E1   +22.346, E3 +529338.636}
ENDSPLINE

SPLINE
SPL {X  -162.820, Y  +621.304, Z    +0.000, E1   +22.259, E3 +529351.452}
SPL {X  -162.820, Y  +618.758, Z    +0.000, E1   +22.239, E3 +529364.602}
SPL {X  -162.820, Y  +616.062, Z    +0.000, E1   +22.275, E3 +529378.023}
SPL {X  -162.820, Y  +613.536, Z    +0.000, E1   +22.242, E3 +529391.145}
SPL {X  -162.820, Y  +611.128, Z    +0.000, E1   +22.252, E3 +529403.315}
SPL {X  -162.820, Y  +608.428, Z    +0.000, E1   +22.255, E3 +529417.099}
SPL {X  -162.820, Y  +605.984, Z    +0.000, E1   +22.221, E3 +529429.735}
SPL {X  -162.820, Y  +603.020, Z    +0.000, E1   +22.272, E3 +529444.634}
SPL {X  -162.820, Y  +599.168, Z    +0.000, E1   +22.310, E3 +529463.902}
SPL {X  -162.820, Y  +595.597, Z    +0.000, E1   +22.284, E3 +529482.238}
SPL {X  -162.820, Y  +593.320, Z    +0.000, E1   +22.199, E3 +529494.328}
SPL {X  -162.820, Y  +591.031, Z    +0.000, E1   +22.283, E3 +529505.419}
SPL {X  -162.820, Y  +588.026, Z    +0.000, E1   +22.301, E3 +529520.546}
SPL {X  -162.820, Y  +585.899, Z    +0.000, E1   +22.286, E3 +529531.348}
SPL {X  -162.820, Y  +583.204, Z    +0.000, E1   +22.278, E3 +529545.371}
SPL {X  -162.820, Y  +579.691, Z    +0.000, E1   +22.312, E3 +529562.859}
SPL {X  -162.820, Y  +577.460, Z    +0.000, E1   +22.218, E3 +529574.846}
SPL {X  -162.820, Y  +575.394, Z    +0.000, E1   +22.240, E3 +529585.271}
SPL {X  -162.820, Y  +572.645, Z    +0.000, E1   +22.246, E3 +529599.269}
SPL {X  -162.820, Y  +570.282, Z    +0.000, E1   +22.231, E3 +529611.319}
SPL {X  -162.820, Y  +567.961, Z    +0.000, E1   +22.247, E3 +529623.109}
SPL {X  -162.820, Y  +564.506, Z    +0.000, E1   +22.298, E3 +529640.423}
SPL {X  -162.820, Y  +561.620, Z    +0.000, E1   +22.191, E3 +529655.804}
SPL {X  -162.820, Y  +559.515, Z    +0.000, E1   +22.273, E3 +529665.806}
SPL {X  -162.820, Y  +556.723, Z    +0.000, E1   +22.309, E3 +529679.889}
SPL {X  -162.820, Y  +554.378, Z    +0.000, E1   +22.288, E3 +529691.735}
SPL {X  -162.820, Y  +552.787, Z    +0.000, E1   +22.213, E3 +529700.557}
SPL {X  -162.820, Y  +550.871, Z    +0.000, E1   +22.229, E3 +529710.151}
SPL {X  -162.820, Y  +548.168, Z    +0.000, E1   +22.298, E3 +529723.487}
SPL {X  -162.820, Y  +545.860, Z    +0.000, E1   +22.216, E3 +529735.745}
SPL {X  -162.820, Y  +543.558, Z    +0.000, E1   +22.285, E3 +529746.975}
SPL {X  -162.820, Y  +540.968, Z    +0.000, E1   +22.274, E3 +529760.248}
SPL {X  -162.820, Y  +538.512, Z    +0.000, E1   +22.287, E3 +529772.560}
SPL {X  -162.820, Y  +535.523, Z    +0.000, E1   +22.266, E3 +529788.176}
SPL {X  -162.820, Y  +531.757, Z    +0.000, E1   +22.276, E3 +529807.230}
SPL {X  -162.820, Y  +527.980, Z    +0.000, E1   +22.326, E3 +529826.061}
SPL {X  -162.820, Y  +524.599, Z    +0.000, E1   +22.287, E3 +529843.459}
SPL {X  -162.820, Y  +522.011, Z    +0.000, E1   +22.282, E3 +529856.535}
SPL {X  -162.820, Y  +519.457, Z    +0.000, E1   +22.481, E3 +529867.825}
SPL {X  -162.820, Y  +505.859, Z    +0.000, E1   +28.367, E3 +529882.308}
SPL {X  -162.820, Y  +504.131, Z    +0.000, E1   +27.325, E3 +529896.446}
SPL {X  -162.820, Y  +503.215, Z    +0.000, E1   +26.369, E3 +529907.132}
SPL {X  -162.820, Y  +502.265, Z    +0.000, E1   +25.287, E3 +529919.614}
SPL {X  -162.820, Y  +501.060, Z    +0.000, E1   +24.081, E3 +529934.355}
SPL {X  -162.820, Y  +500.336, Z    +0.000, E1   +23.110, E3 +529945.495}
SPL {X  -162.820, Y  +499.240, Z    +0.000, E1   +22.316, E3 +529957.805}
SPL {X  -162.820, Y  +498.027, Z    +0.000, E1   +21.516, E3 +529970.713}
SPL {X  -162.820, Y  +495.897, Z    +0.000, E1   +21.662, E3 +529980.633}
SPL {X  -162.820, Y  +493.717, Z    +0.000, E1   +21.704, E3 +529991.740}
SPL {X  -162.820, Y  +491.396, Z    +0.000, E1   +21.707, E3 +530003.864}
SPL {X  -162.820, Y  +488.560, Z    +0.000, E1   +21.695, E3 +530018.973}
SPL {X  -162.820, Y  +485.661, Z    +0.000, E1   +21.712, E3 +530033.858}
SPL {X  -162.820, Y  +483.668, Z    +0.000, E1   +21.664, E3 +530044.686}
SPL {X  -162.820, Y  +481.739, Z    +0.000, E1   +21.704, E3 +530054.400}
SPL {X  -162.820, Y  +479.894, Z    +0.000, E1   +21.695, E3 +530064.187}
SPL {X  -162.820, Y  +477.685, Z    +0.000, E1   +21.656, E3 +530076.124}
SPL {X  -162.820, Y  +475.419, Z    +0.000, E1   +21.711, E3 +530087.477}
SPL {X  -162.820, Y  +473.301, Z    +0.000, E1   +21.712, E3 +530098.574}
SPL {X  -162.820, Y  +470.965, Z    +0.000, E1   +21.700, E3 +530110.919}
SPL {X  -162.820, Y  +469.036, Z    +0.000, E1   +21.695, E3 +530120.963}
SPL {X  -162.820, Y  +467.138, Z    +0.000, E1   +21.678, E3 +530131.134}
SPL {X  -162.820, Y  +465.011, Z    +0.000, E1   +21.692, E3 +530142.117}
SPL {X  -162.820, Y  +462.669, Z    +0.000, E1   +21.752, E3 +530153.898}
SPL {X  -162.820, Y  +460.725, Z    +0.000, E1   +21.689, E3 +530164.511}
SPL {X  -162.820, Y  +458.666, Z    +0.000, E1   +21.695, E3 +530175.323}
SPL {X  -162.820, Y  +456.431, Z    +0.000, E1   +21.708, E3 +530186.851}
SPL {X  -162.820, Y  +454.628, Z    +0.000, E1   +21.674, E3 +530196.569}
SPL {X  -162.820, Y  +452.690, Z    +0.000, E1   +21.773, E3 +530205.843}
SPL {X  -162.820, Y  +450.610, Z    +0.000, E1   +21.698, E3 +530217.442}
SPL {X  -162.820, Y  +448.170, Z    +0.000, E1   +21.667, E3 +530230.463}
SPL {X  -162.820, Y  +446.246, Z    +0.000, E1   +21.696, E3 +530240.281}
SPL {X  -162.820, Y  +443.784, Z    +0.000, E1   +21.713, E3 +530253.067}
SPL {X  -162.820, Y  +440.567, Z    +0.000, E1   +21.731, E3 +530269.907}
SPL {X  -162.820, Y  +437.628, Z    +0.000, E1   +21.678, E3 +530285.571}
SPL {X  -162.820, Y  +435.262, Z    +0.000, E1   +21.727, E3 +530297.507}
SPL {X  -162.820, Y  +433.510, Z    +0.000, E1   +21.692, E3 +530306.920}
SPL {X  -162.820, Y  +431.492, Z    +0.000, E1   +21.686, E3 +530317.616}
SPL {X  -162.820, Y  +429.074, Z    +0.000, E1   +21.710, E3 +530330.068}
SPL {X  -162.820, Y  +427.020, Z    +0.000, E1   +21.674, E3 +530341.069}
SPL {X  -162.820, Y  +424.525, Z    +0.000, E1   +21.712, E3 +530353.982}
SPL {X  -162.820, Y  +421.144, Z    +0.000, E1   +21.719, E3 +530371.649}
SPL {X  -162.820, Y  +418.116, Z    +0.000, E1   +21.761, E3 +530386.980}
SPL {X  -162.820, Y  +416.127, Z    +0.000, E1   +21.715, E3 +530397.686}
SPL {X  -162.820, Y  +414.361, Z    +0.000, E1   +21.613, E3 +530407.873}
SPL {X  -162.820, Y  +412.134, Z    +0.000, E1   +21.697, E3 +530418.817}
SPL {X  -162.820, Y  +409.248, Z    +0.000, E1   +21.741, E3 +530433.753}
SPL {X  -162.820, Y  +406.238, Z    +0.000, E1   +21.697, E3 +530449.721}
SPL {X  -162.820, Y  +404.001, Z    +0.000, E1   +21.723, E3 +530461.150}
SPL {X  -162.820, Y  +402.223, Z    +0.000, E1   +21.697, E3 +530470.636}
SPL {X  -162.820, Y  +400.348, Z    +0.000, E1   +21.713, E3 +530480.361}
SPL {X  -162.820, Y  +398.298, Z    +0.000, E1   +21.721, E3 +530490.977}
SPL {X  -162.820, Y  +396.371, Z    +0.000, E1   +21.713, E3 +530501.159}
SPL {X  -162.820, Y  +394.508, Z    +0.000, E1   +21.616, E3 +530511.714}
SPL {X  -162.820, Y  +392.435, Z    +0.000, E1   +21.681, E3 +530522.068}
SPL {X  -162.820, Y  +389.390, Z    +0.000, E1   +21.742, E3 +530537.674}
SPL {X  -162.820, Y  +386.818, Z    +0.000, E1   +21.679, E3 +530551.433}
SPL {X  -162.820, Y  +384.697, Z    +0.000, E1   +21.693, E3 +530562.503}
SPL {X  -162.820, Y  +382.288, Z    +0.000, E1   +21.742, E3 +530574.627}
SPL {X  -162.817, Y  +379.520, Z    +0.000, E1   +21.723, E3 +530589.464}
SPL {X  -162.776, Y  +376.710, Z    +0.000, E1   +21.698, E3 +530604.204}
SPL {X  -162.707, Y  +374.438, Z    +0.000, E1   +21.688, E3 +530616.207}
SPL {X  -162.607, Y  +372.171, Z    +0.000, E1   +21.692, E3 +530628.007}
SPL {X  -162.494, Y  +370.197, Z    +0.000, E1   +21.655, E3 +530638.633}
SPL {X  -162.349, Y  +368.131, Z    +0.000, E1   +21.624, E3 +530649.751}
SPL {X  -162.161, Y  +365.866, Z    +0.000, E1   +21.642, E3 +530661.437}
SPL {X  -161.927, Y  +363.466, Z    +0.000, E1   +21.730, E3 +530673.208}
SPL {X  -160.290, Y  +351.907, Z    +0.000, E1   +27.562, E3 +530680.786}
SPL {X  -160.281, Y  +351.857, Z    +0.000, E1   +24.243, E3 +530710.199}
ENDSPLINE

SPLINE
SPL {X  -161.833, Y  +362.603, Z    +0.000, E1   +17.021, E3 +530724.895}
ENDSPLINE

SPLINE
SPL {X  -160.786, Y  +354.842, Z    +0.000, E1   +19.274, E3 +530757.050}
ENDSPLINE

SPLINE
SPL {X  -162.485, Y  +370.062, Z    +0.000, E1   +10.606, E3 +530763.429}
SPL {X  -162.818, Y  +379.636, Z    +0.000, E1    +5.115, E3 +530752.777}
SPL {X  -162.820, Y  +386.976, Z    +0.000, E1    +0.144, E3 +530751.876}
SPL {X  -162.820, Y  +391.982, Z    +0.000, E1    -3.443, E3 +530758.641}
SPL {X  -162.820, Y  +399.630, Z    +0.000, E1    -9.426, E3 +530761.149}
SPL {X  -162.820, Y  +408.127, Z    +0.000, E1   -18.417, E3 +530747.437}
SPL {X  -162.820, Y  +420.083, Z    +0.000, E1   -24.325, E3 +530767.913}
SPL {X  -162.820, Y  +428.527, Z    +0.000, E1   -26.988, E3 +530785.205}
SPL {X  -162.820, Y  +431.336, Z    +0.000, E1   -24.162, E3 +530815.415}
SPL {X  -162.820, Y  +432.048, Z    +0.000, E1   -22.832, E3 +530829.919}
SPL {X  -162.820, Y  +434.888, Z    +0.000, E1   -22.823, E3 +530843.868}
SPL {X  -162.820, Y  +436.834, Z    +0.000, E1   -22.779, E3 +530853.828}
SPL {X  -162.820, Y  +438.868, Z    +0.000, E1   -22.837, E3 +530863.482}
SPL {X  -162.820, Y  +441.351, Z    +0.000, E1   -22.805, E3 +530876.057}
SPL {X  -162.820, Y  +443.809, Z    +0.000, E1   -22.804, E3 +530888.223}
SPL {X  -162.820, Y  +447.077, Z    +0.000, E1   -22.869, E3 +530904.034}
SPL {X  -162.820, Y  +449.911, Z    +0.000, E1   -22.774, E3 +530918.643}
SPL {X  -162.820, Y  +451.861, Z    +0.000, E1   -22.750, E3 +530928.491}
SPL {X  -162.820, Y  +454.167, Z    +0.000, E1   -22.842, E3 +530939.220}
SPL {X  -162.820, Y  +456.529, Z    +0.000, E1   -22.855, E3 +530950.749}
SPL {X  -162.820, Y  +458.725, Z    +0.000, E1   -22.793, E3 +530962.153}
SPL {X  -162.820, Y  +461.700, Z    +0.000, E1   -22.822, E3 +530976.775}
SPL {X  -162.820, Y  +464.633, Z    +0.000, E1   -22.813, E3 +530991.272}
SPL {X  -162.820, Y  +466.699, Z    +0.000, E1   -22.824, E3 +531001.318}
SPL {X  -162.820, Y  +468.655, Z    +0.000, E1   -22.858, E3 +531010.762}
SPL {X  -162.820, Y  +470.892, Z    +0.000, E1   -22.837, E3 +531022.001}
SPL {X  -162.820, Y  +473.485, Z    +0.000, E1   -22.806, E3 +531035.199}
SPL {X  -162.820, Y  +475.738, Z    +0.000, E1   -22.728, E3 +531046.864}
SPL {X  -162.820, Y  +478.177, Z    +0.000, E1   -22.834, E3 +531058.204}
SPL {X  -162.820, Y  +481.034, Z    +0.000, E1   -22.831, E3 +531072.341}
SPL {X  -162.820, Y  +483.391, Z    +0.000, E1   -22.793, E3 +531084.277}
SPL {X  -162.820, Y  +486.307, Z    +0.000, E1   -22.833, E3 +531098.531}
SPL {X  -162.820, Y  +489.750, Z    +0.000, E1   -22.832, E3 +531115.601}
SPL {X  -162.820, Y  +492.546, Z    +0.000, E1   -22.823, E3 +531129.359}
SPL {X  -162.820, Y  +495.526, Z    +0.000, E1   -22.833, E3 +531144.242}
SPL {X  -162.820, Y  +499.330, Z    +0.000, E1   -22.841, E3 +531163.023}
SPL {X  -162.820, Y  +503.049, Z    +0.000, E1   -22.823, E3 +531181.573}
SPL {X  -162.820, Y  +506.908, Z    +0.000, E1   -22.877, E3 +531200.242}
SPL {X  -162.820, Y  +510.068, Z    +0.000, E1   -22.761, E3 +531216.714}
SPL {X  -162.820, Y  +512.359, Z    +0.000, E1   -22.823, E3 +531227.446}
SPL {X  -162.820, Y  +513.873, Z    +0.000, E1   -22.800, E3 +531235.132}
SPL {X  -162.820, Y  +516.100, Z    +0.000, E1   -22.809, E3 +531246.209}
SPL {X  -162.820, Y  +518.662, Z    +0.000, E1   -22.847, E3 +531258.507}
SPL {X  -162.820, Y  +520.641, Z    +0.000, E1   -22.790, E3 +531268.748}
SPL {X  -162.820, Y  +523.535, Z    +0.000, E1   -22.857, E3 +531282.717}
SPL {X  -162.820, Y  +526.661, Z    +0.000, E1   -22.801, E3 +531298.541}
SPL {X  -162.820, Y  +528.725, Z    +0.000, E1   -22.770, E3 +531308.911}
SPL {X  -162.820, Y  +530.303, Z    +0.000, E1   -22.798, E3 +531316.530}
SPL {X  -162.820, Y  +532.614, Z    +0.000, E1   -22.828, E3 +531327.798}
SPL {X  -162.820, Y  +534.838, Z    +0.000, E1   -22.864, E3 +531338.427}
SPL {X  -162.820, Y  +536.882, Z    +0.000, E1   -22.782, E3 +531349.282}
SPL {X  -162.820, Y  +539.194, Z    +0.000, E1   -22.826, E3 +531360.330}
SPL {X  -162.820, Y  +541.555, Z    +0.000, E1   -22.817, E3 +531372.145}
SPL {X  -162.820, Y  +543.728, Z    +0.000, E1   -22.799, E3 +531383.002}
SPL {X  -162.820, Y  +545.925, Z    +0.000, E1   -22.803, E3 +531393.872}
SPL {X  -162.820, Y  +549.071, Z    +0.000, E1   -22.836, E3 +531409.400}
SPL {X  -162.820, Y  +553.089, Z    +0.000, E1   -22.838, E3 +531429.300}
SPL {X  -162.820, Y  +556.430, Z    +0.000, E1   -22.821, E3 +531445.801}
SPL {X  -162.820, Y  +559.675, Z    +0.000, E1   -22.837, E3 +531461.881}
SPL {X  -162.820, Y  +562.799, Z    +0.000, E1   -22.814, E3 +531477.387}
SPL {X  -162.820, Y  +565.170, Z    +0.000, E1   -22.801, E3 +531489.212}
SPL {X  -162.820, Y  +568.020, Z    +0.000, E1   -22.787, E3 +531503.599}
SPL {X  -162.820, Y  +570.992, Z    +0.000, E1   -22.834, E3 +531517.818}
SPL {X  -162.820, Y  +572.901, Z    +0.000, E1   -22.775, E3 +531527.686}
SPL {X  -162.820, Y  +575.638, Z    +0.000, E1   -22.855, E3 +531540.796}
SPL {X  -162.820, Y  +578.553, Z    +0.000, E1   -22.801, E3 +531555.508}
SPL {X  -162.820, Y  +581.064, Z    +0.000, E1   -22.823, E3 +531567.793}
SPL {X  -162.820, Y  +583.435, Z    +0.000, E1   -22.808, E3 +531579.614}
SPL {X  -162.820, Y  +585.410, Z    +0.000, E1   -22.764, E3 +531589.750}
SPL {X  -162.820, Y  +587.676, Z    +0.000, E1   -22.853, E3 +531600.265}
SPL {X  -162.820, Y  +589.682, Z    +0.000, E1   -22.776, E3 +531610.794}
SPL {X  -162.820, Y  +591.720, Z    +0.000, E1   -22.868, E3 +531620.105}
SPL {X  -162.820, Y  +593.650, Z    +0.000, E1   -22.810, E3 +531630.175}
SPL {X  -162.820, Y  +595.830, Z    +0.000, E1   -22.828, E3 +531640.791}
SPL {X  -162.820, Y  +598.094, Z    +0.000, E1   -22.843, E3 +531651.904}
SPL {X  -162.820, Y  +600.420, Z    +0.000, E1   -22.826, E3 +531663.535}
SPL {X  -162.820, Y  +602.573, Z    +0.000, E1   -22.830, E3 +531674.121}
SPL {X  -162.820, Y  +604.828, Z    +0.000, E1   -22.784, E3 +531685.759}
SPL {X  -162.820, Y  +608.133, Z    +0.000, E1   -22.831, E3 +531701.877}
SPL {X  -162.820, Y  +611.103, Z    +0.000, E1   -22.785, E3 +531716.802}
SPL {X  -162.820, Y  +613.294, Z    +0.000, E1   -22.780, E3 +531727.676}
SPL {X  -162.820, Y  +615.356, Z    +0.000, E1   -22.799, E3 +531737.733}
SPL {X  -162.820, Y  +617.439, Z    +0.000, E1   -22.808, E3 +531747.991}
SPL {X  -162.820, Y  +619.665, Z    +0.000, E1   -22.817, E3 +531758.959}
SPL {X  -162.820, Y  +621.733, Z    +0.000, E1   -22.759, E3 +531769.683}
SPL {X  -162.820, Y  +624.076, Z    +0.000, E1   -22.774, E3 +531781.188}
SPL {X  -162.820, Y  +627.244, Z    +0.000, E1   -22.803, E3 +531796.871}
SPL {X  -162.820, Y  +630.349, Z    +0.000, E1   -22.766, E3 +531812.402}
SPL {X  -162.820, Y  +632.572, Z    +0.000, E1   -22.785, E3 +531823.209}
SPL {X  -162.820, Y  +634.507, Z    +0.000, E1   -22.784, E3 +531832.848}
SPL {X  -162.820, Y  +636.863, Z    +0.000, E1   -22.760, E3 +531844.770}
SPL {X  -162.820, Y  +640.111, Z    +0.000, E1   -22.809, E3 +531860.653}
SPL {X  -162.820, Y  +643.449, Z    +0.000, E1   -22.796, E3 +531877.170}
SPL {X  -162.820, Y  +645.630, Z    +0.000, E1   -22.795, E3 +531887.867}
SPL {X  -162.820, Y  +647.561, Z    +0.000, E1   -22.705, E3 +531898.317}
SPL {X  -162.820, Y  +649.758, Z    +0.000, E1   -22.780, E3 +531908.507}
SPL {X  -162.820, Y  +651.708, Z    +0.000, E1   -22.810, E3 +531918.002}
SPL {X  -162.820, Y  +653.898, Z    +0.000, E1   -22.796, E3 +531928.923}
SPL {X  -162.820, Y  +656.161, Z    +0.000, E1   -22.812, E3 +531940.044}
SPL {X  -162.820, Y  +658.384, Z    +0.000, E1   -22.822, E3 +531950.910}
SPL {X  -162.820, Y  +660.215, Z    +0.000, E1   -22.649, E3 +531961.501}
SPL {X  -162.820, Y  +662.823, Z    +0.000, E1   -22.799, E3 +531973.209}
SPL {X  -162.820, Y  +665.112, Z    +0.000, E1   -22.835, E3 +531984.263}
SPL {X  -162.820, Y  +667.016, Z    +0.000, E1   -22.823, E3 +531993.692}
SPL {X  -162.820, Y  +668.960, Z    +0.000, E1   -22.773, E3 +532003.859}
SPL {X  -162.820, Y  +672.333, Z    +0.000, E1   -22.837, E3 +532020.195}
SPL {X  -162.812, Y  +675.071, Z    +0.000, E1   -22.742, E3 +532034.340}
SPL {X  -162.773, Y  +677.428, Z    +0.000, E1   -22.762, E3 +532045.938}
SPL {X  -162.691, Y  +679.987, Z    +0.000, E1   -22.794, E3 +532058.351}
SPL {X  -162.604, Y  +681.880, Z    +0.000, E1   -22.691, E3 +532068.512}
SPL {X  -162.458, Y  +684.346, Z    +0.000, E1   -22.764, E3 +532080.305}
SPL {X  -162.296, Y  +686.547, Z    +0.000, E1   -22.660, E3 +532091.922}
SPL {X  -162.090, Y  +688.902, Z    +0.000, E1   -22.700, E3 +532103.430}
SPL {X  -161.474, Y  +694.390, Z    +0.000, E1   -24.298, E3 +532116.786}
SPL {X  -158.730, Y  +709.763, Z    +0.000, E1   -31.225, E3 +532128.124}
ENDSPLINE

SPLINE
SPL {X  -160.932, Y  +698.225, Z    +0.000, E1   -21.712, E3 +532159.234}
SPL {X  -161.691, Y  +692.643, Z    +0.000, E1   -17.369, E3 +532176.116}
SPL {X  -162.534, Y  +683.153, Z    +0.000, E1   -10.475, E3 +532201.583}
SPL {X  -162.820, Y  +667.630, Z    +0.000, E1    -0.882, E3 +532195.560}
SPL {X  -162.820, Y  +661.883, Z    +0.000, E1    +3.373, E3 +532201.003}
SPL {X  -162.820, Y  +653.808, Z    +0.000, E1    +9.891, E3 +532198.694}
SPL {X  -162.820, Y  +632.548, Z    +0.000, E1   +27.446, E3 +532195.231}
ENDSPLINE

SPLINE
SPL {X  -162.820, Y  +638.080, Z    +0.000, E1   +18.858, E3 +532222.979}
ENDSPLINE

SPLINE
SPL {X  -162.820, Y  +623.278, Z    +0.000, E1   +28.723, E3 +532224.550}
SPL {X  -162.820, Y  +618.658, Z    +0.000, E1   +26.841, E3 +532253.159}
ENDSPLINE

SPLINE
SPL {X  -162.820, Y  +623.685, Z    +0.000, E1   +22.346, E3 +532265.466}
ENDSPLINE

SPLINE
SPL {X  -162.820, Y  +621.304, Z    +0.000, E1   +22.259, E3 +532278.281}
SPL {X  -162.820, Y  +618.758, Z    +0.000, E1   +22.239, E3 +532291.432}
SPL {X  -162.820, Y  +616.062, Z    +0.000, E1   +22.275, E3 +532304.852}
SPL {X  -162.820, Y  +613.536, Z    +0.000, E1   +22.242, E3 +532317.974}
SPL {X  -162.820, Y  +611.128, Z    +0.000, E1   +22.252, E3 +532330.145}
SPL {X  -162.820, Y  +608.428, Z    +0.000, E1   +22.255, E3 +532343.928}
SPL {X  -162.820, Y  +605.178, Z    +0.000, E1   +22.267, E3 +532360.460}
SPL {X  -162.820, Y  +602.350, Z    +0.000, E1   +22.224, E3 +532375.077}
SPL {X  -162.820, Y  +599.842, Z    +0.000, E1   +22.298, E3 +532387.229}
SPL {X  -162.820, Y  +597.194, Z    +0.000, E1   +22.253, E3 +532401.150}
SPL {X  -162.820, Y  +594.779, Z    +0.000, E1   +22.284, E3 +532413.054}
SPL {X  -162.820, Y  +592.389, Z    +0.000, E1   +22.245, E3 +532425.670}
SPL {X  -162.820, Y  +589.492, Z    +0.000, E1   +22.304, E3 +532439.855}
SPL {X  -162.820, Y  +587.447, Z    +0.000, E1   +22.279, E3 +532450.383}
SPL {X  -162.820, Y  +585.192, Z    +0.000, E1   +22.298, E3 +532461.794}
SPL {X  -162.820, Y  +582.610, Z    +0.000, E1   +22.234, E3 +532475.417}
SPL {X  -162.820, Y  +580.317, Z    +0.000, E1   +22.300, E3 +532486.471}
SPL {X  -162.820, Y  +578.878, Z    +0.000, E1   +22.272, E3 +532493.980}
SPL {X  -162.820, Y  +576.856, Z    +0.000, E1   +22.233, E3 +532504.739}
SPL {X  -162.820, Y  +574.811, Z    +0.000, E1   +22.236, E3 +532515.002}
SPL {X  -162.820, Y  +572.645, Z    +0.000, E1   +22.246, E3 +532526.098}
SPL {X  -162.820, Y  +569.475, Z    +0.000, E1   +22.269, E3 +532542.104}
SPL {X  -162.820, Y  +565.838, Z    +0.000, E1   +22.271, E3 +532560.699}
SPL {X  -162.820, Y  +562.162, Z    +0.000, E1   +22.252, E3 +532579.516}
SPL {X  -162.820, Y  +558.919, Z    +0.000, E1   +22.286, E3 +532595.679}
SPL {X  -162.820, Y  +556.169, Z    +0.000, E1   +22.295, E3 +532609.509}
SPL {X  -162.820, Y  +553.294, Z    +0.000, E1   +22.266, E3 +532624.506}
SPL {X  -162.820, Y  +550.136, Z    +0.000, E1   +22.258, E3 +532640.619}
SPL {X  -162.820, Y  +546.694, Z    +0.000, E1   +22.290, E3 +532657.942}
SPL {X  -162.820, Y  +543.558, Z    +0.000, E1   +22.285, E3 +532673.804}
SPL {X  -162.820, Y  +541.633, Z    +0.000, E1   +22.257, E3 +532683.733}
SPL {X  -162.820, Y  +539.116, Z    +0.000, E1   +22.302, E3 +532696.343}
SPL {X  -162.820, Y  +536.913, Z    +0.000, E1   +22.192, E3 +532708.268}
SPL {X  -162.820, Y  +534.880, Z    +0.000, E1   +22.252, E3 +532718.221}
SPL {X  -162.820, Y  +532.896, Z    +0.000, E1   +22.234, E3 +532728.382}
SPL {X  -162.820, Y  +531.056, Z    +0.000, E1   +22.251, E3 +532737.663}
SPL {X  -162.820, Y  +528.708, Z    +0.000, E1   +22.319, E3 +532749.045}
SPL {X  -162.820, Y  +525.932, Z    +0.000, E1   +22.258, E3 +532763.801}
SPL {X  -162.820, Y  +522.524, Z    +0.000, E1   +22.326, E3 +532780.525}
SPL {X  -162.820, Y  +519.457, Z    +0.000, E1   +22.481, E3 +532794.654}
SPL {X  -162.820, Y  +506.285, Z    +0.000, E1   +28.538, E3 +532806.112}
SPL {X  -162.820, Y  +504.441, Z    +0.000, E1   +27.574, E3 +532820.454}
SPL {X  -162.820, Y  +503.215, Z    +0.000, E1   +26.369, E3 +532833.961}
SPL {X  -162.820, Y  +502.265, Z    +0.000, E1   +25.287, E3 +532846.444}
SPL {X  -162.820, Y  +501.060, Z    +0.000, E1   +24.081, E3 +532861.184}
SPL {X  -162.820, Y  +500.336, Z    +0.000, E1   +23.110, E3 +532872.324}
SPL {X  -162.820, Y  +499.240, Z    +0.000, E1   +22.316, E3 +532884.635}
SPL {X  -162.820, Y  +498.027, Z    +0.000, E1   +21.516, E3 +532897.542}
SPL {X  -162.820, Y  +495.897, Z    +0.000, E1   +21.662, E3 +532907.463}
SPL {X  -162.820, Y  +493.717, Z    +0.000, E1   +21.704, E3 +532918.569}
SPL {X  -162.820, Y  +491.396, Z    +0.000, E1   +21.707, E3 +532930.693}
SPL {X  -162.820, Y  +488.560, Z    +0.000, E1   +21.695, E3 +532945.802}
SPL {X  -162.820, Y  +485.661, Z    +0.000, E1   +21.712, E3 +532960.688}
SPL {X  -162.820, Y  +483.668, Z    +0.000, E1   +21.664, E3 +532971.515}
SPL {X  -162.820, Y  +481.739, Z    +0.000, E1   +21.704, E3 +532981.229}
SPL {X  -162.820, Y  +479.894, Z    +0.000, E1   +21.695, E3 +532991.016}
SPL {X  -162.820, Y  +477.685, Z    +0.000, E1   +21.656, E3 +533002.954}
SPL {X  -162.820, Y  +475.419, Z    +0.000, E1   +21.711, E3 +533014.306}
SPL {X  -162.820, Y  +473.301, Z    +0.000, E1   +21.712, E3 +533025.403}
SPL {X  -162.820, Y  +470.965, Z    +0.000, E1   +21.700, E3 +533037.748}
SPL {X  -162.820, Y  +469.036, Z    +0.000, E1   +21.695, E3 +533047.792}
SPL {X  -162.820, Y  +467.138, Z    +0.000, E1   +21.678, E3 +533057.964}
SPL {X  -162.820, Y  +465.011, Z    +0.000, E1   +21.692, E3 +533068.946}
SPL {X  -162.820, Y  +462.669, Z    +0.000, E1   +21.752, E3 +533080.727}
SPL {X  -162.820, Y  +460.725, Z    +0.000, E1   +21.689, E3 +533091.340}
SPL {X  -162.820, Y  +458.666, Z    +0.000, E1   +21.695, E3 +533102.152}
SPL {X  -162.820, Y  +456.431, Z    +0.000, E1   +21.708, E3 +533113.680}
SPL {X  -162.820, Y  +454.628, Z    +0.000, E1   +21.674, E3 +533123.399}
SPL {X  -162.820, Y  +452.690, Z    +0.000, E1   +21.773, E3 +533132.673}
SPL {X  -162.820, Y  +450.610, Z    +0.000, E1   +21.698, E3 +533144.271}
SPL {X  -162.820, Y  +448.170, Z    +0.000, E1   +21.667, E3 +533157.292}
SPL {X  -162.820, Y  +446.246, Z    +0.000, E1   +21.696, E3 +533167.110}
SPL {X  -162.820, Y  +443.784, Z    +0.000, E1   +21.713, E3 +533179.896}
SPL {X  -162.820, Y  +441.754, Z    +0.000, E1   +21.708, E3 +533190.448}
SPL {X  -162.820, Y  +439.933, Z    +0.000, E1   +21.690, E3 +533200.212}
SPL {X  -162.820, Y  +437.628, Z    +0.000, E1   +21.678, E3 +533212.400}
SPL {X  -162.820, Y  +435.262, Z    +0.000, E1   +21.727, E3 +533224.336}
SPL {X  -162.820, Y  +433.510, Z    +0.000, E1   +21.692, E3 +533233.750}
SPL {X  -162.820, Y  +431.492, Z    +0.000, E1   +21.686, E3 +533244.445}
SPL {X  -162.820, Y  +429.074, Z    +0.000, E1   +21.710, E3 +533256.897}
SPL {X  -162.820, Y  +427.020, Z    +0.000, E1   +21.674, E3 +533267.898}
SPL {X  -162.820, Y  +425.215, Z    +0.000, E1   +21.693, E3 +533277.201}
SPL {X  -162.820, Y  +422.986, Z    +0.000, E1   +21.685, E3 +533289.012}
SPL {X  -162.820, Y  +420.528, Z    +0.000, E1   +21.706, E3 +533301.662}
SPL {X  -162.820, Y  +418.116, Z    +0.000, E1   +21.761, E3 +533313.810}
SPL {X  -162.820, Y  +416.127, Z    +0.000, E1   +21.715, E3 +533324.515}
SPL {X  -162.820, Y  +414.361, Z    +0.000, E1   +21.613, E3 +533334.702}
SPL {X  -162.820, Y  +411.450, Z    +0.000, E1   +21.710, E3 +533349.275}
SPL {X  -162.820, Y  +408.590, Z    +0.000, E1   +21.735, E3 +533363.901}
SPL {X  -162.820, Y  +406.238, Z    +0.000, E1   +21.697, E3 +533376.550}
SPL {X  -162.820, Y  +404.001, Z    +0.000, E1   +21.723, E3 +533387.980}
SPL {X  -162.820, Y  +402.223, Z    +0.000, E1   +21.697, E3 +533397.465}
SPL {X  -162.820, Y  +400.348, Z    +0.000, E1   +21.713, E3 +533407.191}
SPL {X  -162.820, Y  +398.298, Z    +0.000, E1   +21.721, E3 +533417.806}
SPL {X  -162.820, Y  +396.371, Z    +0.000, E1   +21.713, E3 +533427.988}
SPL {X  -162.820, Y  +394.508, Z    +0.000, E1   +21.616, E3 +533438.543}
SPL {X  -162.820, Y  +392.435, Z    +0.000, E1   +21.681, E3 +533448.897}
SPL {X  -162.820, Y  +389.390, Z    +0.000, E1   +21.742, E3 +533464.504}
SPL {X  -162.820, Y  +386.818, Z    +0.000, E1   +21.679, E3 +533478.262}
SPL {X  -162.820, Y  +384.697, Z    +0.000, E1   +21.693, E3 +533489.333}
SPL {X  -162.820, Y  +382.288, Z    +0.000, E1   +21.742, E3 +533501.456}
SPL {X  -162.820, Y  +380.381, Z    +0.000, E1   +21.655, E3 +533512.181}
SPL {X  -162.808, Y  +378.512, Z    +0.000, E1   +21.736, E3 +533521.234}
SPL {X  -162.776, Y  +376.710, Z    +0.000, E1   +21.698, E3 +533531.033}
SPL {X  -162.707, Y  +374.438, Z    +0.000, E1   +21.688, E3 +533543.037}
SPL {X  -162.607, Y  +372.171, Z    +0.000, E1   +21.692, E3 +533554.836}
SPL {X  -162.494, Y  +370.197, Z    +0.000, E1   +21.655, E3 +533565.463}
SPL {X  -162.349, Y  +368.131, Z    +0.000, E1   +21.624, E3 +533576.581}
SPL {X  -162.161, Y  +365.866, Z    +0.000, E1   +21.642, E3 +533588.266}
SPL {X  -161.927, Y  +363.466, Z    +0.000, E1   +21.730, E3 +533600.037}
SPL {X  -160.290, Y  +351.907, Z    +0.000, E1   +27.562, E3 +533607.615}
SPL {X  -159.725, Y  +348.905, Z    +0.000, E1   +26.136, E3 +533632.850}
ENDSPLINE

SPLINE
SPL {X  -160.871, Y  +355.385, Z    +0.000, E1   +21.841, E3 +533641.693}
SPL {X  -161.833, Y  +362.603, Z    +0.000, E1   +17.021, E3 +533651.724}
ENDSPLINE

SPLINE
SPL {X  -160.786, Y  +354.842, Z    +0.000, E1   +19.274, E3 +533683.880}
ENDSPLINE

